C09107=1075.584,103.581,430.931,173.685,24.123,154.241
C09108=1075.591,103.830,430.912,173.686,24.125,154.241
C09109=1075.596,104.079,430.894,173.688,24.128,154.241
C09110=1075.601,104.329,430.875,173.690,24.130,154.241
C09111=1075.608,104.578,430.856,173.691,24.133,154.242
C09112=1075.613,104.827,430.838,173.693,24.135,154.242
C09113=1075.618,105.077,430.818,173.695,24.138,154.242
C09114=1075.625,105.326,430.800,173.696,24.141,154.243
C09115=1075.630,105.576,430.781,173.697,24.143,154.243
C09116=1075.635,105.824,430.762,173.700,24.146,154.243
C09117=1075.642,106.074,430.744,173.701,24.148,154.244
C09118=1075.647,106.323,430.724,173.702,24.151,154.244
C09119=1075.653,106.572,430.705,173.705,24.153,154.244
C09120=1075.659,106.821,430.688,173.706,24.156,154.244
C09121=1075.664,107.071,430.668,173.707,24.158,154.245
C09122=1075.669,107.320,430.649,173.710,24.161,154.245
C09123=1075.676,107.569,430.631,173.711,24.163,154.245
C09124=1075.682,107.818,430.612,173.712,24.165,154.246
C09125=1075.687,108.068,430.592,173.715,24.168,154.246
C09126=1075.693,108.316,430.574,173.716,24.171,154.246
C09127=1075.699,108.565,430.555,173.717,24.173,154.246
C09128=1075.704,108.816,430.536,173.720,24.176,154.247
C09129=1075.711,109.065,430.518,173.721,24.178,154.247
C09130=1075.716,109.313,430.499,173.722,24.180,154.247
C09131=1075.721,109.563,430.479,173.724,24.183,154.247
C09132=1075.728,109.812,430.461,173.726,24.185,154.248
C09133=1075.733,110.061,430.442,173.727,24.188,154.248
C09134=1075.739,110.311,430.422,173.729,24.190,154.248
C09135=1075.745,110.559,430.404,173.731,24.193,154.249
C09136=1075.751,110.840,430.382,173.733,24.196,154.249
C09137=1075.758,111.122,430.360,173.735,24.199,154.249
C09138=1075.764,111.404,430.339,173.736,24.202,154.250
C09139=1075.771,111.686,430.318,173.739,24.204,154.250
C09140=1075.777,111.935,430.298,173.740,24.207,154.250
C09141=1075.782,112.184,430.280,173.742,24.210,154.250
C09142=1075.788,112.433,430.261,173.744,24.212,154.251
C09143=1075.794,112.682,430.242,173.745,24.214,154.251
C09144=1075.799,112.932,430.222,173.747,24.217,154.251
C09145=1075.805,113.181,430.203,173.749,24.219,154.252
C09146=1075.810,113.430,430.184,173.750,24.222,154.252
C09147=1075.817,113.679,430.166,173.752,24.224,154.252
C09148=1075.823,113.928,430.146,173.754,24.227,154.252
C09149=1075.828,114.177,430.126,173.755,24.229,154.253
C09150=1075.834,114.427,430.107,173.757,24.232,154.253
C09151=1075.839,114.676,430.088,173.758,24.235,154.253
C09152=1075.845,114.925,430.069,173.761,24.237,154.254
C09153=1075.850,115.174,430.050,173.762,24.240,154.254
C09154=1075.856,115.424,430.030,173.763,24.242,154.254
C09155=1075.861,115.673,430.012,173.766,24.245,154.254
C09156=1075.867,115.921,429.992,173.767,24.247,154.255
C09157=1075.873,116.171,429.972,173.768,24.250,154.255
C09158=1075.879,116.420,429.953,173.771,24.252,154.255
C09159=1075.884,116.670,429.934,173.772,24.255,154.256
C09160=1075.889,116.918,429.915,173.774,24.257,154.256
C09161=1075.895,117.167,429.895,173.776,24.260,154.256
C09162=1075.901,117.417,429.876,173.777,24.263,154.257
C09163=1075.906,117.666,429.856,173.779,24.265,154.257
C09164=1075.912,117.916,429.837,173.780,24.268,154.257
C09165=1075.917,118.164,429.817,173.783,24.270,154.257
C09166=1075.923,118.413,429.798,173.784,24.273,154.258
C09167=1075.928,118.663,429.779,173.785,24.275,154.258
C09168=1075.934,118.912,429.759,173.788,24.278,154.258
C09169=1075.940,119.161,429.739,173.789,24.280,154.259
C09170=1075.946,119.410,429.720,173.790,24.282,154.259
C09171=1075.952,119.660,429.701,173.793,24.285,154.259
C09172=1075.957,119.908,429.681,173.794,24.288,154.259
C09173=1075.963,120.157,429.662,173.796,24.290,154.260
C09174=1075.968,120.407,429.643,173.798,24.293,154.260
C09175=1075.973,120.657,429.623,173.799,24.295,154.260
C09176=1075.979,120.905,429.603,173.801,24.298,154.260
C09177=1075.985,121.155,429.584,173.803,24.300,154.261
C09178=1075.991,121.404,429.564,173.805,24.303,154.261
C09179=1075.997,121.653,429.545,173.806,24.305,154.261
C09180=1076.002,121.903,429.525,173.808,24.307,154.262
C09181=1076.008,122.151,429.506,173.810,24.310,154.262
C09182=1076.013,122.400,429.487,173.811,24.312,154.262
C09183=1076.019,122.649,429.467,173.814,24.315,154.262
C09184=1076.024,122.899,429.447,173.815,24.318,154.263
C09185=1076.030,123.148,429.428,173.817,24.320,154.263
C09186=1076.036,123.397,429.408,173.819,24.323,154.263
C09187=1076.042,123.646,429.388,173.820,24.325,154.264
C09188=1076.048,123.895,429.368,173.822,24.328,154.264
C09189=1076.053,124.145,429.349,173.824,24.330,154.264
C09190=1076.059,124.393,429.329,173.826,24.333,154.264
C09191=1076.064,124.643,429.309,173.827,24.335,154.265
C09192=1076.070,124.892,429.289,173.829,24.337,154.265
C09193=1076.076,125.141,429.270,173.831,24.340,154.265
C09194=1076.082,125.390,429.250,173.832,24.342,154.265
C09195=1076.088,125.640,429.231,173.835,24.345,154.266
C09196=1076.094,125.888,429.211,173.836,24.347,154.266
C09197=1076.099,126.138,429.191,173.838,24.350,154.266
C09198=1076.105,126.387,429.171,173.840,24.353,154.267
C09199=1076.110,126.636,429.152,173.841,24.355,154.267
C09200=1076.117,126.917,429.130,173.843,24.358,154.267
C09201=1076.123,127.199,429.107,173.846,24.360,154.267
C09202=1076.130,127.481,429.085,173.848,24.363,154.268
C09203=1076.136,127.761,429.063,173.849,24.366,154.268
C09204=1076.141,128.011,429.043,173.851,24.369,154.268
C09205=1076.147,128.260,429.023,173.853,24.371,154.269
C09206=1076.154,128.509,429.003,173.855,24.373,154.269
C09207=1076.160,128.759,428.983,173.856,24.375,154.269
C09208=1076.166,129.008,428.963,173.859,24.378,154.269
C09209=1076.171,129.257,428.943,173.860,24.381,154.270
C09210=1076.177,129.506,428.924,173.861,24.383,154.270
C09211=1076.183,129.755,428.904,173.864,24.386,154.270
C09212=1076.189,130.004,428.884,173.865,24.388,154.270
C09213=1076.194,130.253,428.864,173.867,24.391,154.271
C09214=1076.199,130.502,428.844,173.869,24.392,154.271
C09215=1076.205,130.751,428.824,173.871,24.395,154.271
C09216=1076.211,131.001,428.805,173.873,24.397,154.271
C09217=1076.217,131.249,428.785,173.875,24.400,154.272
C09218=1076.223,131.499,428.764,173.876,24.402,154.272
C09219=1076.229,131.748,428.744,173.879,24.405,154.272
C09220=1076.235,131.998,428.725,173.880,24.407,154.272
C09221=1076.241,132.246,428.705,173.881,24.409,154.273
C09222=1076.246,132.495,428.684,173.884,24.412,154.273
C09223=1076.252,132.744,428.664,173.885,24.414,154.273
C09224=1076.257,132.994,428.644,173.887,24.417,154.273
C09225=1076.263,133.243,428.624,173.889,24.419,154.274
C09226=1076.268,133.492,428.604,173.891,24.422,154.274
C09227=1076.274,133.741,428.584,173.892,24.424,154.274
C09228=1076.279,133.990,428.563,173.895,24.427,154.275
C09229=1076.285,134.239,428.544,173.896,24.430,154.275
C09230=1076.290,134.488,428.523,173.898,24.432,154.275
C09231=1076.297,134.738,428.503,173.900,24.435,154.275
C09232=1076.302,134.987,428.483,173.902,24.437,154.276
C09233=1076.308,135.236,428.463,173.903,24.440,154.276
C09234=1076.313,135.485,428.442,173.905,24.442,154.276
C09235=1076.319,135.734,428.422,173.907,24.444,154.276
C09236=1076.325,135.983,428.402,173.909,24.446,154.277
C09237=1076.330,136.232,428.382,173.911,24.449,154.277
C09238=1076.336,136.482,428.362,173.912,24.451,154.277
C09239=1076.342,136.731,428.341,173.915,24.454,154.277
C09240=1076.347,136.980,428.321,173.916,24.456,154.278
C09241=1076.353,137.229,428.301,173.918,24.459,154.278
C09242=1076.359,137.478,428.280,173.920,24.462,154.278
C09243=1076.365,137.727,428.260,173.922,24.464,154.279
C09244=1076.370,137.976,428.240,173.923,24.466,154.279
C09245=1076.376,138.225,428.220,173.926,24.469,154.279
C09246=1076.382,138.475,428.199,173.927,24.471,154.279
C09247=1076.388,138.724,428.179,173.929,24.474,154.280
C09248=1076.393,138.973,428.158,173.931,24.476,154.280
C09249=1076.399,139.221,428.138,173.933,24.479,154.280
C09250=1076.404,139.471,428.118,173.934,24.481,154.280
C09251=1076.410,139.720,428.097,173.937,24.484,154.281
C09252=1076.416,139.969,428.077,173.938,24.486,154.281
C09253=1076.421,140.218,428.057,173.940,24.488,154.281
C09254=1076.427,140.467,428.037,173.942,24.491,154.281
C09255=1076.433,140.716,428.016,173.944,24.493,154.282
C09256=1076.438,140.965,427.995,173.945,24.496,154.282
C09257=1076.444,141.215,427.974,173.948,24.498,154.282
C09258=1076.450,141.463,427.954,173.949,24.501,154.282
C09259=1076.455,141.713,427.933,173.951,24.503,154.283
C09260=1076.461,141.962,427.913,173.953,24.506,154.283
C09261=1076.467,142.210,427.893,173.955,24.508,154.283
C09262=1076.472,142.460,427.872,173.956,24.511,154.284
C09263=1076.478,142.709,427.851,173.959,24.513,154.284
C09264=1076.484,142.990,427.828,173.961,24.516,154.284
C09265=1076.491,143.271,427.804,173.963,24.519,154.284
C09266=1076.497,143.552,427.781,173.965,24.521,154.285
C09267=1076.503,143.834,427.758,173.967,24.524,154.285
C09268=1076.509,144.083,427.738,173.969,24.527,154.285
C09269=1076.515,144.333,427.717,173.971,24.529,154.285
C09270=1076.520,144.582,427.696,173.973,24.532,154.286
C09271=1076.526,144.830,427.675,173.974,24.534,154.286
C09272=1076.532,145.079,427.655,173.977,24.537,154.286
C09273=1076.538,145.329,427.634,173.978,24.539,154.287
C09274=1076.543,145.578,427.614,173.980,24.542,154.287
C09275=1076.548,145.827,427.592,173.982,24.543,154.287
C09276=1076.554,146.076,427.572,173.984,24.546,154.287
C09277=1076.560,146.325,427.551,173.986,24.549,154.288
C09278=1076.566,146.574,427.530,173.988,24.551,154.288
C09279=1076.571,146.823,427.510,173.990,24.554,154.288
C09280=1076.577,147.073,427.489,173.992,24.556,154.288
C09281=1076.583,147.321,427.468,173.994,24.558,154.288
C09282=1076.588,147.570,427.448,173.995,24.561,154.289
C09283=1076.594,147.820,427.427,173.998,24.563,154.289
C09284=1076.600,148.068,427.405,173.999,24.566,154.289
C09285=1076.605,148.318,427.385,174.001,24.568,154.290
C09286=1076.610,148.567,427.364,174.003,24.571,154.290
C09287=1076.617,148.816,427.343,174.005,24.573,154.290
C09288=1076.623,149.065,427.323,174.007,24.575,154.290
C09289=1076.628,149.313,427.301,174.009,24.578,154.291
C09290=1076.634,149.563,427.280,174.011,24.581,154.291
C09291=1076.639,149.812,427.260,174.013,24.583,154.291
C09292=1076.645,150.061,427.239,174.015,24.586,154.291
C09293=1076.651,150.310,427.218,174.016,24.588,154.292
C09294=1076.656,150.559,427.196,174.019,24.590,154.292
C09295=1076.661,150.808,427.176,174.020,24.592,154.292
C09296=1076.668,151.057,427.154,174.022,24.595,154.292
C09297=1076.673,151.306,427.134,174.025,24.598,154.293
C09298=1076.678,151.555,427.112,174.026,24.600,154.293
C09299=1076.684,151.805,427.091,174.028,24.603,154.293
C09300=1076.690,152.053,427.070,174.030,24.605,154.293
C09301=1076.695,152.302,427.050,174.032,24.607,154.294
C09302=1076.701,152.552,427.028,174.034,24.610,154.294
C09303=1076.707,152.801,427.007,174.036,24.612,154.294
C09304=1076.712,153.049,426.986,174.038,24.615,154.294
C09305=1076.718,153.299,426.965,174.040,24.617,154.295
C09306=1076.724,153.548,426.944,174.042,24.620,154.295
C09307=1076.730,153.797,426.922,174.043,24.622,154.295
C09308=1076.735,154.046,426.902,174.046,24.624,154.295
C09309=1076.741,154.294,426.881,174.047,24.627,154.296
C09310=1076.746,154.544,426.860,174.049,24.629,154.296
C09311=1076.752,154.793,426.838,174.052,24.632,154.296
C09312=1076.758,155.042,426.817,174.053,24.634,154.297
C09313=1076.763,155.291,426.796,174.055,24.637,154.297
C09314=1076.769,155.540,426.775,174.057,24.639,154.297
C09315=1076.774,155.789,426.753,174.059,24.642,154.297
C09316=1076.780,156.038,426.732,174.061,24.644,154.297
C09317=1076.786,156.287,426.710,174.063,24.647,154.298
C09318=1076.791,156.536,426.689,174.065,24.649,154.298
C09319=1076.797,156.785,426.669,174.067,24.651,154.298
C09320=1076.803,157.034,426.647,174.069,24.654,154.298
C09321=1076.808,157.283,426.626,174.071,24.656,154.299
C09322=1076.814,157.532,426.604,174.073,24.659,154.299
C09323=1076.819,157.781,426.583,174.075,24.661,154.299
C09324=1076.825,158.031,426.561,174.076,24.664,154.300
C09325=1076.831,158.279,426.540,174.079,24.666,154.300
C09326=1076.837,158.528,426.518,174.081,24.669,154.300
C09327=1076.842,158.777,426.498,174.083,24.671,154.300
C09328=1076.848,159.059,426.473,174.085,24.674,154.301
C09329=1076.855,159.339,426.449,174.087,24.676,154.301
C09330=1076.861,159.620,426.425,174.089,24.679,154.301
C09331=1076.868,159.902,426.401,174.092,24.682,154.301
C09332=1076.873,160.150,426.379,174.094,24.684,154.302
C09333=1076.879,160.399,426.358,174.095,24.687,154.302
C09334=1076.884,160.648,426.336,174.098,24.689,154.302
C09335=1076.890,160.898,426.315,174.100,24.692,154.302
C09336=1076.896,161.146,426.294,174.101,24.694,154.303
C09337=1076.902,161.396,426.272,174.104,24.696,154.303
C09338=1076.906,161.644,426.250,174.106,24.699,154.303
C09339=1076.913,161.894,426.229,174.108,24.701,154.303
C09340=1076.917,162.142,426.207,174.110,24.704,154.304
C09341=1076.924,162.392,426.185,174.111,24.706,154.304
C09342=1076.928,162.640,426.163,174.114,24.709,154.304
C09343=1076.935,162.890,426.142,174.116,24.712,154.304
C09344=1076.939,163.138,426.120,174.117,24.714,154.305
C09345=1076.946,163.388,426.098,174.120,24.717,154.305
C09346=1076.950,163.636,426.076,174.122,24.719,154.305
C09347=1076.956,163.885,426.055,174.123,24.722,154.306
C09348=1076.961,164.135,426.033,174.126,24.724,154.306
C09349=1076.967,164.383,426.011,174.128,24.727,154.306
C09350=1076.972,164.633,425.989,174.129,24.729,154.306
C09351=1076.978,164.881,425.968,174.132,24.732,154.307
C09352=1076.983,165.131,425.946,174.134,24.734,154.307
C09353=1076.989,165.379,425.924,174.136,24.736,154.307
C09354=1076.994,165.629,425.902,174.138,24.739,154.307
C09355=1077.000,165.877,425.881,174.140,24.742,154.308
C09356=1077.005,166.127,425.859,174.142,24.744,154.308
C09357=1077.011,166.375,425.837,174.144,24.747,154.308
C09358=1077.016,166.625,425.815,174.146,24.749,154.308
C09359=1077.021,166.873,425.793,174.148,24.752,154.309
C09360=1077.028,167.122,425.771,174.150,24.754,154.309
C09361=1077.033,167.372,425.749,174.152,24.757,154.309
C09362=1077.039,167.620,425.727,174.154,24.759,154.309
C09363=1077.044,167.870,425.705,174.156,24.762,154.310
C09364=1077.050,168.118,425.684,174.158,24.764,154.310
C09365=1077.055,168.368,425.662,174.160,24.767,154.310
C09366=1077.060,168.616,425.640,174.162,24.769,154.310
C09367=1077.066,168.865,425.618,174.164,24.772,154.311
C09368=1077.072,169.114,425.595,174.166,24.774,154.311
C09369=1077.077,169.363,425.574,174.168,24.776,154.311
C09370=1077.083,169.613,425.552,174.171,24.779,154.311
C09371=1077.089,169.860,425.530,174.172,24.781,154.312
C09372=1077.094,170.110,425.508,174.174,24.784,154.312
C09373=1077.099,170.359,425.485,174.177,24.787,154.312
C09374=1077.105,170.608,425.464,174.179,24.789,154.313
C09375=1077.111,170.857,425.441,174.180,24.791,154.313
C09376=1077.116,171.105,425.420,174.183,24.794,154.313
C09377=1077.122,171.355,425.398,174.185,24.796,154.313
C09378=1077.127,171.604,425.375,174.186,24.799,154.314
C09379=1077.133,171.852,425.353,174.189,24.801,154.314
C09380=1077.138,172.102,425.331,174.191,24.804,154.314
C09381=1077.144,172.351,425.309,174.193,24.806,154.314
C09382=1077.150,172.599,425.287,174.195,24.809,154.314
C09383=1077.155,172.849,425.265,174.197,24.811,154.315
C09384=1077.162,173.097,425.242,174.200,24.814,154.315
C09385=1077.166,173.346,425.221,174.201,24.816,154.315
C09386=1077.172,173.596,425.198,174.203,24.818,154.315
C09387=1077.178,173.844,425.176,174.206,24.821,154.316
C09388=1077.184,174.094,425.154,174.207,24.823,154.316
C09389=1077.189,174.342,425.131,174.209,24.826,154.316
C09390=1077.195,174.591,425.110,174.212,24.829,154.317
C09391=1077.201,174.841,425.087,174.214,24.831,154.317
C09392=1077.206,175.121,425.062,174.216,24.834,154.317
C09393=1077.213,175.401,425.037,174.219,24.837,154.317
C09394=1077.219,175.682,425.011,174.221,24.839,154.318
C09395=1077.226,175.963,424.987,174.223,24.842,154.318
C09396=1077.232,176.212,424.964,174.226,24.845,154.318
C09397=1077.237,176.460,424.942,174.228,24.847,154.318
C09398=1077.242,176.710,424.920,174.230,24.849,154.319
C09399=1077.249,176.958,424.897,174.232,24.852,154.319
C09400=1077.254,177.208,424.875,174.234,24.854,154.319
C09401=1077.260,177.457,424.852,174.236,24.856,154.319
C09402=1077.266,177.705,424.831,174.238,24.859,154.319
C09403=1077.271,177.954,424.808,174.240,24.861,154.320
C09404=1077.277,178.204,424.786,174.243,24.864,154.320
C09405=1077.283,178.452,424.763,174.245,24.866,154.320
C09406=1077.289,178.701,424.740,174.247,24.869,154.320
C09407=1077.294,178.950,424.718,174.249,24.871,154.321
C09408=1077.299,179.199,424.695,174.251,24.874,154.321
C09409=1077.306,179.448,424.674,174.254,24.876,154.321
C09410=1077.311,179.697,424.651,174.255,24.878,154.321
C09411=1077.317,179.946,424.628,174.257,24.881,154.322
C09412=1077.323,180.195,424.606,174.260,24.884,154.322
C09413=1077.328,180.443,424.584,174.262,24.886,154.322
C09414=1077.334,180.692,424.561,174.264,24.888,154.322
C09415=1077.340,180.942,424.539,174.266,24.891,154.323
C09416=1077.345,181.191,424.516,174.268,24.893,154.323
C09417=1077.352,181.439,424.493,174.271,24.895,154.323
C09418=1077.357,181.688,424.470,174.273,24.898,154.323
C09419=1077.363,181.938,424.448,174.275,24.900,154.323
C09420=1077.369,182.187,424.425,174.277,24.903,154.324
C09421=1077.375,182.434,424.403,174.279,24.905,154.324
C09422=1077.380,182.683,424.380,174.282,24.908,154.324
C09423=1077.386,182.933,424.358,174.284,24.910,154.324
C09424=1077.391,183.182,424.335,174.285,24.912,154.325
C09425=1077.397,183.431,424.312,174.288,24.915,154.325
C09426=1077.404,183.679,424.290,174.290,24.917,154.325
C09427=1077.409,183.928,424.267,174.293,24.920,154.325
C09428=1077.415,184.178,424.245,174.295,24.922,154.326
C09429=1077.420,184.427,424.222,174.296,24.924,154.326
C09430=1077.426,184.675,424.199,174.299,24.927,154.326
C09431=1077.433,184.924,424.176,174.301,24.929,154.326
C09432=1077.438,185.173,424.153,174.303,24.932,154.327
C09433=1077.443,185.421,424.130,174.306,24.935,154.327
C09434=1077.449,185.670,424.107,174.307,24.937,154.327
C09435=1077.454,185.919,424.084,174.310,24.939,154.327
C09436=1077.460,186.169,424.062,174.312,24.942,154.328
C09437=1077.465,186.418,424.039,174.314,24.945,154.328
C09438=1077.470,186.667,424.016,174.317,24.947,154.328
C09439=1077.476,186.915,423.993,174.318,24.949,154.328
C09440=1077.481,187.164,423.970,174.320,24.952,154.329
C09441=1077.487,187.413,423.947,174.323,24.955,154.329
C09442=1077.493,187.662,423.924,174.325,24.957,154.329
C09443=1077.498,187.911,423.901,174.327,24.960,154.329
C09444=1077.503,188.160,423.878,174.330,24.963,154.330
C09445=1077.509,188.409,423.855,174.331,24.965,154.330
C09446=1077.515,188.658,423.832,174.334,24.967,154.330
C09447=1077.519,188.906,423.809,174.336,24.970,154.330
C09448=1077.525,189.155,423.786,174.338,24.972,154.331
C09449=1077.531,189.403,423.762,174.341,24.975,154.331
C09450=1077.537,189.652,423.739,174.343,24.978,154.331
C09451=1077.543,189.901,423.716,174.345,24.980,154.331
C09452=1077.548,190.150,423.693,174.347,24.983,154.332
C09453=1077.553,190.399,423.670,174.349,24.985,154.332
C09454=1077.559,190.648,423.647,174.351,24.988,154.332
C09455=1077.565,190.897,423.624,174.354,24.990,154.332
C09456=1077.571,191.177,423.597,174.356,24.993,154.333
C09457=1077.577,191.458,423.571,174.358,24.996,154.333
C09458=1077.583,191.739,423.545,174.362,24.999,154.333
C09459=1077.589,192.018,423.519,174.364,25.002,154.334
C09460=1077.594,192.267,423.496,174.366,25.004,154.334
C09461=1077.600,192.516,423.473,174.369,25.007,154.334
C09462=1077.606,192.764,423.449,174.370,25.009,154.334
C09463=1077.612,193.013,423.426,174.372,25.012,154.335
C09464=1077.617,193.262,423.402,174.375,25.014,154.335
C09465=1077.623,193.511,423.380,174.377,25.017,154.335
C09466=1077.629,193.760,423.355,174.379,25.019,154.335
C09467=1077.634,194.010,423.332,174.382,25.022,154.336
C09468=1077.640,194.258,423.309,174.384,25.025,154.336
C09469=1077.646,194.507,423.286,174.386,25.027,154.336
C09470=1077.651,194.756,423.262,174.389,25.030,154.336
C09471=1077.657,195.005,423.239,174.390,25.032,154.337
C09472=1077.662,195.254,423.216,174.392,25.035,154.337
C09473=1077.668,195.502,423.192,174.395,25.037,154.337
C09474=1077.673,195.751,423.169,174.397,25.039,154.337
C09475=1077.679,196.000,423.146,174.400,25.042,154.338
C09476=1077.685,196.248,423.122,174.402,25.045,154.338
C09477=1077.690,196.498,423.099,174.404,25.047,154.338
C09478=1077.696,196.747,423.076,174.407,25.050,154.338
C09479=1077.701,196.995,423.051,174.409,25.052,154.339
C09480=1077.707,197.244,423.028,174.411,25.055,154.339
C09481=1077.714,197.493,423.004,174.413,25.057,154.339
C09482=1077.719,197.742,422.981,174.415,25.060,154.339
C09483=1077.725,197.990,422.957,174.418,25.062,154.340
C09484=1077.730,198.239,422.934,174.420,25.064,154.340
C09485=1077.735,198.489,422.911,174.422,25.067,154.340
C09486=1077.741,198.737,422.887,174.425,25.070,154.340
C09487=1077.747,198.986,422.864,174.427,25.072,154.341
C09488=1077.753,199.235,422.839,174.429,25.075,154.341
C09489=1077.759,199.484,422.817,174.432,25.078,154.341
C09490=1077.764,199.733,422.792,174.434,25.080,154.341
C09491=1077.770,199.981,422.769,174.437,25.082,154.342
C09492=1077.776,200.230,422.746,174.439,25.085,154.342
C09493=1077.781,200.478,422.721,174.441,25.088,154.342
C09494=1077.787,200.728,422.698,174.444,25.090,154.342
C09495=1077.793,200.976,422.674,174.446,25.092,154.343
C09496=1077.798,201.225,422.651,174.447,25.095,154.343
C09497=1077.805,201.474,422.627,174.450,25.097,154.343
C09498=1077.810,201.723,422.604,174.452,25.100,154.343
C09499=1077.816,201.972,422.580,174.454,25.103,154.344
C09500=1077.821,202.220,422.555,174.457,25.105,154.344
C09501=1077.827,202.469,422.532,174.459,25.107,154.344
C09502=1077.832,202.718,422.508,174.462,25.110,154.344
C09503=1077.839,202.967,422.484,174.464,25.113,154.345
C09504=1077.844,203.216,422.461,174.466,25.115,154.345
C09505=1077.849,203.465,422.436,174.469,25.118,154.345
C09506=1077.855,203.713,422.413,174.471,25.121,154.345
C09507=1077.860,203.962,422.389,174.473,25.123,154.346
C09508=1077.866,204.211,422.365,174.476,25.126,154.346
C09509=1077.872,204.460,422.341,174.478,25.129,154.346
C09510=1077.878,204.708,422.317,174.480,25.131,154.346
C09511=1077.883,204.958,422.293,174.483,25.134,154.347
C09512=1077.889,205.206,422.269,174.485,25.136,154.347
C09513=1077.895,205.455,422.245,174.487,25.139,154.347
C09514=1077.900,205.704,422.221,174.490,25.141,154.347
C09515=1077.906,205.952,422.197,174.492,25.144,154.348
C09516=1077.911,206.201,422.173,174.495,25.146,154.348
C09517=1077.916,206.450,422.149,174.497,25.149,154.348
C09518=1077.922,206.699,422.124,174.499,25.152,154.348
C09519=1077.928,206.947,422.101,174.502,25.154,154.349
C09520=1077.956,208.196,421.979,174.611,25.215,154.348
C09521=1077.962,208.408,421.958,174.614,25.218,154.349
C09522=1077.967,208.620,421.937,174.616,25.221,154.349
C09523=1077.971,208.832,421.917,174.617,25.224,154.349
C09524=1077.976,209.045,421.895,174.619,25.227,154.350
C09525=1077.981,209.257,421.874,174.621,25.230,154.350
C09526=1077.986,209.470,421.853,174.623,25.233,154.351
C09527=1077.991,209.681,421.832,174.625,25.236,154.351
C09528=1077.997,209.931,421.807,174.627,25.239,154.352
C09529=1078.002,210.180,421.783,174.629,25.243,154.352
C09530=1078.008,210.428,421.758,174.631,25.247,154.353
C09531=1078.014,210.677,421.733,174.633,25.250,154.353
C09532=1078.020,210.925,421.708,174.636,25.254,154.354
C09533=1078.025,211.175,421.683,174.639,25.258,154.354
C09534=1078.030,211.423,421.658,174.641,25.261,154.354
C09535=1078.036,211.672,421.633,174.643,25.264,154.355
C09536=1078.042,211.920,421.608,174.645,25.268,154.356
C09537=1078.048,212.169,421.584,174.647,25.271,154.356
C09538=1078.053,212.417,421.559,174.649,25.275,154.356
C09539=1078.059,212.667,421.534,174.651,25.279,154.357
C09540=1078.065,212.915,421.509,174.654,25.282,154.357
C09541=1078.071,213.164,421.485,174.656,25.285,154.358
C09542=1078.076,213.413,421.459,174.659,25.289,154.358
C09543=1078.082,213.661,421.434,174.661,25.293,154.359
C09544=1078.088,213.910,421.409,174.663,25.296,154.359
C09545=1078.094,214.159,421.384,174.665,25.300,154.360
C09546=1078.098,214.408,421.359,174.667,25.304,154.360
C09547=1078.105,214.656,421.333,174.669,25.307,154.361
C09548=1078.110,214.904,421.309,174.671,25.310,154.361
C09549=1078.116,215.154,421.284,174.673,25.314,154.362
C09550=1078.122,215.402,421.258,174.676,25.318,154.362
C09551=1078.127,215.650,421.233,174.679,25.321,154.363
C09552=1078.133,215.900,421.208,174.681,25.325,154.363
C09553=1078.139,216.148,421.183,174.683,25.329,154.364
C09554=1078.144,216.397,421.157,174.685,25.332,154.364
C09555=1078.150,216.646,421.133,174.687,25.335,154.365
C09556=1078.156,216.894,421.108,174.689,25.339,154.365
C09557=1078.162,217.143,421.083,174.692,25.343,154.366
C09558=1078.167,217.392,421.057,174.695,25.346,154.366
C09559=1078.173,217.640,421.032,174.697,25.350,154.367
C09560=1078.178,217.878,421.007,174.699,25.353,154.367
C09561=1078.184,218.117,420.984,174.701,25.357,154.368
C09562=1078.189,218.356,420.960,174.703,25.360,154.368
C09563=1078.195,218.594,420.935,174.705,25.363,154.368
C09564=1078.201,218.834,420.910,174.707,25.367,154.369
C09565=1078.206,219.072,420.887,174.710,25.370,154.369
C09566=1078.212,219.311,420.862,174.712,25.373,154.370
C09567=1078.217,219.550,420.837,174.714,25.377,154.370
C09568=1078.223,219.797,420.812,174.716,25.380,154.371
C09569=1078.229,220.046,420.787,174.718,25.384,154.371
C09570=1078.234,220.295,420.761,174.721,25.387,154.372
C09571=1078.241,220.544,420.736,174.723,25.391,154.372
C09572=1078.246,220.792,420.712,174.726,25.395,154.373
C09573=1078.251,221.041,420.686,174.728,25.398,154.373
C09574=1078.258,221.290,420.660,174.730,25.401,154.374
C09575=1078.264,221.539,420.635,174.732,25.405,154.374
C09576=1078.273,221.947,420.593,174.737,25.411,154.375
C09577=1078.282,222.356,420.550,174.740,25.417,154.376
C09578=1078.291,222.764,420.508,174.744,25.423,154.376
C09579=1078.300,223.173,420.467,174.747,25.428,154.377
C09580=1078.306,223.422,420.441,174.749,25.432,154.378
C09581=1078.312,223.671,420.416,174.752,25.436,154.378
C09582=1078.318,223.920,420.390,174.755,25.439,154.379
C09583=1078.323,224.167,420.364,174.757,25.443,154.379
C09584=1078.329,224.416,420.338,174.759,25.446,154.380
C09585=1078.335,224.665,420.313,174.761,25.450,154.380
C09586=1078.341,224.914,420.287,174.764,25.453,154.381
C09587=1078.346,225.163,420.261,174.766,25.457,154.381
C09588=1078.352,225.411,420.236,174.768,25.461,154.382
C09589=1078.357,225.660,420.210,174.771,25.464,154.382
C09590=1078.364,225.908,420.184,174.773,25.467,154.383
C09591=1078.369,226.157,420.158,174.776,25.471,154.383
C09592=1078.375,226.406,420.132,174.778,25.474,154.383
C09593=1078.381,226.654,420.107,174.780,25.478,154.384
C09594=1078.386,226.903,420.081,174.782,25.482,154.384
C09595=1078.392,227.151,420.055,174.784,25.485,154.385
C09596=1078.398,227.400,420.029,174.787,25.489,154.385
C09597=1078.403,227.649,420.003,174.790,25.493,154.386
C09598=1078.410,227.897,419.977,174.792,25.496,154.386
C09599=1078.415,228.146,419.951,174.794,25.499,154.387
C09600=1078.421,228.395,419.925,174.796,25.502,154.387
C09601=1078.427,228.643,419.900,174.799,25.506,154.388
C09602=1078.433,228.892,419.873,174.801,25.510,154.388
C09603=1078.439,229.140,419.848,174.804,25.513,154.389
C09604=1078.444,229.389,419.822,174.806,25.517,154.389
C09605=1078.449,229.637,419.796,174.809,25.521,154.390
C09606=1078.456,229.886,419.770,174.811,25.524,154.390
C09607=1078.461,230.134,419.744,174.813,25.528,154.391
C09608=1078.467,230.383,419.718,174.815,25.531,154.391
C09609=1078.472,230.632,419.692,174.818,25.535,154.392
C09610=1078.478,230.880,419.665,174.820,25.538,154.392
C09611=1078.484,231.129,419.640,174.823,25.542,154.393
C09612=1078.490,231.377,419.613,174.825,25.545,154.393
C09613=1078.496,231.626,419.587,174.827,25.549,154.394
C09614=1078.501,231.875,419.561,174.830,25.553,154.394
C09615=1078.507,232.124,419.535,174.832,25.556,154.394
C09616=1078.513,232.372,419.508,174.834,25.559,154.395
C09617=1078.519,232.621,419.483,174.836,25.563,154.395
C09618=1078.525,232.869,419.456,174.840,25.567,154.396
C09619=1078.530,233.118,419.430,174.842,25.570,154.396
C09620=1078.536,233.366,419.403,174.844,25.574,154.397
C09621=1078.542,233.615,419.377,174.846,25.577,154.397
C09622=1078.547,233.864,419.351,174.849,25.581,154.398
C09623=1078.553,234.112,419.324,174.851,25.585,154.398
C09624=1078.558,234.360,419.299,174.853,25.588,154.399
C09625=1078.563,234.609,419.272,174.856,25.591,154.399
C09626=1078.569,234.857,419.245,174.859,25.595,154.400
C09627=1078.575,235.106,419.219,174.861,25.599,154.400
C09628=1078.584,235.507,419.177,174.864,25.604,154.401
C09629=1078.593,235.906,419.134,174.868,25.610,154.402
C09630=1078.603,236.306,419.092,174.873,25.616,154.403
C09631=1078.613,236.707,419.049,174.876,25.622,154.403
C09632=1078.618,236.956,419.022,174.878,25.625,154.404
C09633=1078.624,237.205,418.996,174.882,25.629,154.404
C09634=1078.630,237.453,418.970,174.884,25.632,154.405
C09635=1078.635,237.701,418.943,174.886,25.636,154.405
C09636=1078.641,237.950,418.916,174.888,25.639,154.406
C09637=1078.646,238.198,418.889,174.891,25.643,154.406
C09638=1078.652,238.447,418.863,174.893,25.647,154.407
C09639=1078.657,238.696,418.836,174.895,25.650,154.407
C09640=1078.663,238.944,418.810,174.898,25.654,154.408
C09641=1078.669,239.193,418.783,174.901,25.657,154.408
C09642=1078.675,239.441,418.757,174.903,25.661,154.409
C09643=1078.681,239.690,418.730,174.905,25.664,154.409
C09644=1078.687,239.938,418.703,174.908,25.668,154.410
C09645=1078.693,240.187,418.676,174.910,25.671,154.410
C09646=1078.699,240.435,418.650,174.912,25.675,154.411
C09647=1078.704,240.684,418.624,174.916,25.679,154.411
C09648=1078.710,240.932,418.597,174.918,25.682,154.411
C09649=1078.716,241.181,418.570,174.920,25.686,154.412
C09650=1078.721,241.429,418.543,174.922,25.689,154.412
C09651=1078.727,241.678,418.516,174.925,25.693,154.413
C09652=1078.733,241.927,418.489,174.927,25.696,154.413
C09653=1078.738,242.175,418.463,174.930,25.699,154.414
C09654=1078.744,242.424,418.436,174.933,25.703,154.414
C09655=1078.750,242.671,418.409,174.935,25.707,154.415
C09656=1078.757,242.920,418.382,174.937,25.710,154.415
C09657=1078.762,243.169,418.355,174.940,25.714,154.416
C09658=1078.768,243.417,418.328,174.942,25.718,154.416
C09659=1078.773,243.666,418.301,174.944,25.721,154.417
C09660=1078.778,243.914,418.274,174.948,25.725,154.417
C09661=1078.784,244.163,418.247,174.950,25.728,154.418
C09662=1078.790,244.412,418.220,174.952,25.732,154.418
C09663=1078.796,244.661,418.193,174.955,25.736,154.419
C09664=1078.802,244.908,418.166,174.957,25.739,154.419
C09665=1078.807,245.157,418.139,174.959,25.743,154.420
C09666=1078.812,245.405,418.112,174.961,25.746,154.420
C09667=1078.818,245.654,418.085,174.965,25.750,154.421
C09668=1078.825,245.903,418.058,174.967,25.753,154.421
C09669=1078.830,246.151,418.030,174.969,25.757,154.422
C09670=1078.836,246.399,418.004,174.972,25.761,154.422
C09671=1078.841,246.647,417.977,174.974,25.764,154.423
C09672=1078.847,246.896,417.949,174.976,25.768,154.423
C09673=1078.853,247.145,417.922,174.979,25.772,154.424
C09674=1078.858,247.393,417.895,174.982,25.775,154.424
C09675=1078.864,247.642,417.868,174.985,25.779,154.424
C09676=1078.870,247.890,417.840,174.987,25.782,154.425
C09677=1078.876,248.139,417.813,174.989,25.786,154.426
C09678=1078.881,248.387,417.785,174.992,25.790,154.426
C09679=1078.886,248.635,417.758,174.994,25.793,154.427
C09680=1078.896,249.029,417.714,174.998,25.799,154.427
C09681=1078.905,249.423,417.672,175.003,25.805,154.428
C09682=1078.913,249.816,417.628,175.006,25.811,154.429
C09683=1078.923,250.210,417.585,175.010,25.816,154.430
C09684=1078.928,250.458,417.557,175.013,25.820,154.430
C09685=1078.933,250.707,417.530,175.015,25.824,154.431
C09686=1078.940,250.955,417.502,175.017,25.827,154.431
C09687=1078.945,251.204,417.475,175.021,25.831,154.432
C09688=1078.951,251.452,417.447,175.023,25.834,154.432
C09689=1078.956,251.700,417.420,175.025,25.838,154.433
C09690=1078.962,251.949,417.392,175.028,25.842,154.433
C09691=1078.968,252.197,417.365,175.030,25.845,154.434
C09692=1078.973,252.445,417.337,175.032,25.848,154.434
C09693=1078.979,252.694,417.309,175.035,25.852,154.435
C09694=1078.985,252.942,417.282,175.038,25.856,154.435
C09695=1078.991,253.191,417.254,175.041,25.860,154.436
C09696=1078.997,253.439,417.227,175.043,25.863,154.436
C09697=1079.002,253.688,417.199,175.045,25.867,154.437
C09698=1079.008,253.936,417.171,175.048,25.871,154.437
C09699=1079.014,254.184,417.144,175.050,25.874,154.438
C09700=1079.019,254.433,417.116,175.053,25.878,154.438
C09701=1079.025,254.682,417.088,175.056,25.881,154.439
C09702=1079.031,254.929,417.061,175.058,25.885,154.439
C09703=1079.036,255.179,417.033,175.061,25.889,154.440
C09704=1079.042,255.427,417.005,175.063,25.892,154.440
C09705=1079.048,255.674,416.978,175.066,25.896,154.440
C09706=1079.054,255.923,416.949,175.068,25.899,154.441
C09707=1079.059,256.172,416.922,175.071,25.903,154.442
C09708=1079.065,256.420,416.894,175.074,25.907,154.442
C09709=1079.071,256.668,416.866,175.076,25.910,154.442
C09710=1079.077,256.917,416.838,175.079,25.914,154.443
C09711=1079.082,257.165,416.810,175.081,25.917,154.444
C09712=1079.089,257.414,416.782,175.083,25.921,154.444
C09713=1079.094,257.662,416.755,175.087,25.924,154.444
C09714=1079.100,257.911,416.727,175.089,25.928,154.445
C09715=1079.106,258.159,416.700,175.092,25.932,154.445
C09716=1079.112,258.408,416.671,175.094,25.935,154.446
C09717=1079.117,258.656,416.643,175.096,25.939,154.446
C09718=1079.123,258.904,416.615,175.099,25.943,154.447
C09719=1079.129,259.152,416.588,175.101,25.946,154.447
C09720=1079.135,259.401,416.559,175.105,25.950,154.448
C09721=1079.140,259.649,416.531,175.107,25.953,154.448
C09722=1079.146,259.898,416.503,175.110,25.957,154.449
C09723=1079.152,260.145,416.476,175.112,25.960,154.449
C09724=1079.158,260.394,416.447,175.114,25.964,154.450
C09725=1079.164,260.643,416.419,175.117,25.968,154.450
C09726=1079.170,260.891,416.391,175.120,25.971,154.451
C09727=1079.176,261.139,416.363,175.123,25.975,154.451
C09728=1079.182,261.387,416.335,175.125,25.978,154.452
C09729=1079.188,261.636,416.307,175.128,25.982,154.452
C09730=1079.193,261.884,416.279,175.130,25.985,154.453
C09731=1079.199,262.133,416.251,175.134,25.989,154.453
C09732=1079.208,262.523,416.206,175.137,25.994,154.454
C09733=1079.218,262.914,416.162,175.141,26.000,154.455
C09734=1079.227,263.305,416.118,175.146,26.006,154.455
C09735=1079.237,263.696,416.073,175.149,26.012,154.456
C09736=1079.243,263.944,416.045,175.153,26.015,154.457
C09737=1079.249,264.193,416.017,175.155,26.019,154.457
C09738=1079.254,264.441,415.989,175.158,26.023,154.458
C09739=1079.260,264.689,415.960,175.160,26.026,154.458
C09740=1079.266,264.937,415.932,175.163,26.030,154.459
C09741=1079.272,265.186,415.903,175.165,26.033,154.459
C09742=1079.277,265.435,415.874,175.168,26.037,154.460
C09743=1079.282,265.683,415.846,175.171,26.041,154.460
C09744=1079.288,265.931,415.817,175.173,26.044,154.461
C09745=1079.294,266.179,415.789,175.176,26.048,154.461
C09746=1079.300,266.428,415.760,175.178,26.052,154.462
C09747=1079.306,266.676,415.732,175.181,26.056,154.462
C09748=1079.312,266.924,415.703,175.183,26.059,154.463
C09749=1079.317,267.173,415.675,175.187,26.063,154.463
C09750=1079.324,267.421,415.646,175.189,26.066,154.464
C09751=1079.328,267.669,415.617,175.192,26.070,154.464
C09752=1079.334,267.918,415.589,175.194,26.074,154.465
C09753=1079.341,268.166,415.560,175.197,26.078,154.465
C09754=1079.346,268.414,415.532,175.199,26.081,154.466
C09755=1079.352,268.662,415.503,175.202,26.085,154.466
C09756=1079.358,268.911,415.475,175.205,26.088,154.467
C09757=1079.364,269.159,415.446,175.208,26.092,154.467
C09758=1079.369,269.407,415.417,175.210,26.096,154.468
C09759=1079.375,269.655,415.388,175.213,26.100,154.468
C09760=1079.381,269.904,415.359,175.215,26.103,154.469
C09761=1079.387,270.152,415.331,175.218,26.107,154.469
C09762=1079.392,270.400,415.301,175.221,26.111,154.470
C09763=1079.398,270.649,415.273,175.224,26.115,154.470
C09764=1079.404,270.897,415.244,175.226,26.118,154.471
C09765=1079.410,271.144,415.215,175.229,26.121,154.471
C09766=1079.415,271.393,415.187,175.231,26.125,154.472
C09767=1079.422,271.642,415.157,175.234,26.129,154.472
C09768=1079.428,271.890,415.128,175.237,26.133,154.473
C09769=1079.432,272.138,415.100,175.240,26.136,154.473
C09770=1079.439,272.386,415.071,175.242,26.140,154.474
C09771=1079.445,272.634,415.042,175.245,26.144,154.474
C09772=1079.451,272.883,415.013,175.247,26.147,154.475
C09773=1079.456,273.131,414.984,175.250,26.151,154.475
C09774=1079.462,273.379,414.955,175.253,26.155,154.476
C09775=1079.468,273.627,414.926,175.256,26.159,154.477
C09776=1079.473,273.876,414.897,175.258,26.162,154.477
C09777=1079.480,274.124,414.868,175.261,26.166,154.478
C09778=1079.485,274.372,414.839,175.264,26.170,154.478
C09779=1079.491,274.620,414.810,175.266,26.173,154.478
C09780=1079.496,274.869,414.780,175.269,26.177,154.479
C09781=1079.503,275.117,414.751,175.272,26.181,154.480
C09782=1079.508,275.366,414.722,175.275,26.185,154.480
C09783=1079.513,275.613,414.694,175.277,26.188,154.481
C09784=1079.523,276.007,414.647,175.282,26.194,154.481
C09785=1079.532,276.401,414.601,175.285,26.200,154.482
C09786=1079.542,276.795,414.554,175.290,26.206,154.483
C09787=1079.550,277.189,414.507,175.295,26.212,154.484
C09788=1079.557,277.437,414.478,175.297,26.216,154.484
C09789=1079.562,277.685,414.449,175.300,26.220,154.485
C09790=1079.568,277.934,414.420,175.302,26.223,154.485
C09791=1079.573,278.181,414.390,175.305,26.227,154.486
C09792=1079.580,278.429,414.361,175.308,26.231,154.487
C09793=1079.585,278.678,414.332,175.311,26.235,154.487
C09794=1079.591,278.926,414.302,175.314,26.238,154.488
C09795=1079.597,279.175,414.273,175.316,26.242,154.488
C09796=1079.602,279.423,414.243,175.319,26.246,154.489
C09797=1079.609,279.671,414.214,175.321,26.249,154.489
C09798=1079.614,279.920,414.185,175.324,26.253,154.490
C09799=1079.621,280.167,414.155,175.327,26.257,154.490
C09800=1079.626,280.415,414.125,175.330,26.261,154.491
C09801=1079.632,280.664,414.096,175.333,26.265,154.491
C09802=1079.638,280.912,414.067,175.335,26.268,154.492
C09803=1079.644,281.161,414.037,175.338,26.272,154.492
C09804=1079.649,281.408,414.007,175.340,26.276,154.493
C09805=1079.654,281.656,413.977,175.343,26.280,154.493
C09806=1079.661,281.904,413.948,175.346,26.284,154.494
C09807=1079.666,282.153,413.919,175.349,26.287,154.494
C09808=1079.672,282.400,413.888,175.352,26.291,154.495
C09809=1079.677,282.649,413.859,175.354,26.295,154.496
C09810=1079.684,282.897,413.830,175.357,26.299,154.496
C09811=1079.689,283.145,413.799,175.360,26.303,154.497
C09812=1079.695,283.393,413.770,175.362,26.307,154.497
C09813=1079.700,283.642,413.740,175.365,26.311,154.498
C09814=1079.707,283.889,413.710,175.368,26.314,154.498
C09815=1079.713,284.138,413.681,175.371,26.318,154.499
C09816=1079.718,284.386,413.651,175.374,26.322,154.499
C09817=1079.724,284.634,413.621,175.376,26.325,154.500
C09818=1079.729,284.882,413.591,175.379,26.329,154.500
C09819=1079.735,285.130,413.561,175.381,26.333,154.501
C09820=1079.741,285.378,413.532,175.385,26.337,154.502
C09821=1079.747,285.626,413.501,175.388,26.341,154.502
C09822=1079.753,285.875,413.472,175.390,26.345,154.503
C09823=1079.759,286.122,413.441,175.393,26.348,154.503
C09824=1079.764,286.371,413.412,175.395,26.352,154.504
C09825=1079.770,286.619,413.381,175.398,26.356,154.504
C09826=1079.776,286.867,413.352,175.401,26.360,154.505
C09827=1079.782,287.115,413.322,175.404,26.364,154.505
C09828=1079.788,287.363,413.291,175.407,26.368,154.506
C09829=1079.794,287.612,413.261,175.410,26.372,154.506
C09830=1079.800,287.859,413.231,175.412,26.375,154.507
C09831=1079.805,288.108,413.202,175.415,26.379,154.507
C09832=1079.811,288.356,413.171,175.418,26.383,154.508
C09833=1079.818,288.603,413.141,175.420,26.387,154.509
C09834=1079.823,288.852,413.112,175.424,26.391,154.509
C09835=1079.829,289.099,413.081,175.426,26.394,154.510
C09836=1079.838,289.503,413.032,175.431,26.400,154.510
C09837=1079.847,289.907,412.983,175.435,26.407,154.511
C09838=1079.857,290.311,412.934,175.440,26.413,154.512
C09839=1079.867,290.715,412.884,175.444,26.420,154.513
C09840=1079.873,290.963,412.854,175.447,26.423,154.514
C09841=1079.879,291.211,412.824,175.450,26.428,154.514
C09842=1079.885,291.458,412.793,175.453,26.431,154.515
C09843=1079.889,291.707,412.763,175.456,26.435,154.515
C09844=1079.895,291.955,412.733,175.459,26.439,154.516
C09845=1079.902,292.204,412.702,175.461,26.443,154.517
C09846=1079.907,292.451,412.672,175.464,26.447,154.517
C09847=1079.913,292.699,412.641,175.467,26.451,154.518
C09848=1079.919,292.947,412.611,175.470,26.455,154.518
C09849=1079.925,293.195,412.581,175.473,26.459,154.519
C09850=1079.931,293.443,412.550,175.476,26.463,154.519
C09851=1079.937,293.691,412.520,175.478,26.467,154.520
C09852=1079.942,293.939,412.489,175.481,26.470,154.521
C09853=1079.948,294.187,412.458,175.484,26.474,154.521
C09854=1079.954,294.435,412.428,175.486,26.478,154.522
C09855=1079.960,294.683,412.397,175.490,26.482,154.522
C09856=1079.966,294.931,412.367,175.493,26.486,154.523
C09857=1079.972,295.179,412.337,175.495,26.490,154.523
C09858=1079.977,295.427,412.306,175.498,26.494,154.524
C09859=1079.983,295.676,412.275,175.501,26.498,154.524
C09860=1079.989,295.924,412.245,175.504,26.502,154.525
C09861=1079.995,296.171,412.214,175.506,26.506,154.526
C09862=1080.000,296.420,412.183,175.509,26.510,154.526
C09863=1080.007,296.667,412.152,175.513,26.514,154.527
C09864=1080.013,296.915,412.121,175.515,26.517,154.527
C09865=1080.018,297.163,412.091,175.518,26.522,154.528
C09866=1080.024,297.412,412.060,175.521,26.526,154.528
C09867=1080.030,297.660,412.029,175.523,26.530,154.529
C09868=1080.036,297.907,411.998,175.526,26.533,154.530
C09869=1080.041,298.155,411.967,175.529,26.538,154.530
C09870=1080.048,298.404,411.937,175.533,26.542,154.531
C09871=1080.053,298.652,411.906,175.535,26.546,154.531
C09872=1080.059,298.899,411.875,175.538,26.549,154.532
C09873=1080.064,299.147,411.844,175.541,26.554,154.533
C09874=1080.070,299.396,411.813,175.544,26.558,154.533
C09875=1080.076,299.643,411.781,175.546,26.562,154.534
C09876=1080.082,299.891,411.751,175.549,26.566,154.534
C09877=1080.087,300.139,411.720,175.552,26.570,154.535
C09878=1080.093,300.387,411.688,175.555,26.574,154.536
C09879=1080.098,300.635,411.658,175.558,26.578,154.536
C09880=1080.104,300.883,411.626,175.561,26.582,154.537
C09881=1080.110,301.131,411.595,175.564,26.586,154.537
C09882=1080.115,301.379,411.564,175.566,26.590,154.538
C09883=1080.121,301.626,411.533,175.569,26.594,154.539
C09884=1080.127,301.875,411.502,175.572,26.599,154.539
C09885=1080.133,302.122,411.471,175.575,26.603,154.540
C09886=1080.138,302.371,411.440,175.578,26.607,154.540
C09887=1080.144,302.619,411.408,175.581,26.611,154.541
C09888=1080.154,303.037,411.356,175.586,26.618,154.542
C09889=1080.164,303.454,411.303,175.591,26.625,154.543
C09890=1080.174,303.873,411.250,175.595,26.631,154.544
C09891=1080.184,304.291,411.197,175.601,26.639,154.545
C09892=1080.189,304.539,411.166,175.603,26.642,154.546
C09893=1080.195,304.787,411.134,175.606,26.646,154.546
C09894=1080.201,305.034,411.103,175.609,26.651,154.547
C09895=1080.206,305.282,411.072,175.612,26.655,154.548
C09896=1080.213,305.530,411.041,175.615,26.659,154.548
C09897=1080.218,305.778,411.009,175.617,26.663,154.549
C09898=1080.224,306.027,410.978,175.620,26.667,154.550
C09899=1080.230,306.274,410.947,175.624,26.671,154.550
C09900=1080.236,306.522,410.915,175.627,26.675,154.551
C09901=1080.241,306.770,410.883,175.630,26.680,154.551
C09902=1080.248,307.017,410.851,175.632,26.683,154.552
C09903=1080.253,307.266,410.821,175.635,26.688,154.553
C09904=1080.259,307.514,410.789,175.638,26.692,154.553
C09905=1080.265,307.761,410.757,175.641,26.696,154.554
C09906=1080.271,308.009,410.725,175.644,26.700,154.554
C09907=1080.277,308.257,410.693,175.647,26.704,154.555
C09908=1080.283,308.505,410.662,175.650,26.708,154.556
C09909=1080.289,308.753,410.630,175.653,26.712,154.556
C09910=1080.295,309.001,410.599,175.656,26.717,154.557
C09911=1080.301,309.249,410.567,175.659,26.721,154.557
C09912=1080.307,309.496,410.536,175.662,26.725,154.558
C09913=1080.313,309.745,410.504,175.664,26.729,154.559
C09914=1080.319,309.993,410.472,175.667,26.733,154.559
C09915=1080.324,310.240,410.441,175.671,26.737,154.560
C09916=1080.331,310.488,410.409,175.674,26.741,154.560
C09917=1080.337,310.736,410.377,175.677,26.746,154.561
C09918=1080.342,310.984,410.345,175.679,26.750,154.562
C09919=1080.348,311.232,410.313,175.682,26.754,154.562
C09920=1080.355,311.480,410.282,175.685,26.758,154.563
C09921=1080.361,311.727,410.250,175.688,26.762,154.564
C09922=1080.366,311.975,410.218,175.691,26.766,154.564
C09923=1080.372,312.223,410.186,175.694,26.771,154.565
C09924=1080.378,312.471,410.154,175.698,26.775,154.566
C09925=1080.385,312.719,410.122,175.700,26.778,154.566
C09926=1080.391,312.967,410.090,175.703,26.783,154.567
C09927=1080.397,313.215,410.058,175.706,26.787,154.567
C09928=1080.402,313.462,410.026,175.709,26.791,154.568
C09929=1080.408,313.710,409.994,175.712,26.796,154.569
C09930=1080.415,313.958,409.963,175.715,26.799,154.569
C09931=1080.421,314.206,409.931,175.718,26.804,154.570
C09932=1080.426,314.454,409.899,175.721,26.808,154.570
C09933=1080.433,314.702,409.866,175.724,26.812,154.571
C09934=1080.439,314.950,409.834,175.727,26.816,154.572
C09935=1080.445,315.198,409.802,175.730,26.821,154.572
C09936=1080.450,315.445,409.769,175.733,26.825,154.573
C09937=1080.456,315.693,409.737,175.736,26.829,154.574
C09938=1080.462,315.942,409.705,175.739,26.834,154.575
C09939=1080.467,316.188,409.673,175.741,26.838,154.575
C09940=1080.472,316.399,409.645,175.744,26.842,154.576
C09941=1080.477,316.610,409.617,175.747,26.845,154.576
C09942=1080.482,316.821,409.590,175.749,26.849,154.577
C09943=1080.487,317.031,409.563,175.752,26.853,154.577
C09944=1080.492,317.242,409.535,175.754,26.857,154.578
C09945=1080.496,317.453,409.507,175.757,26.860,154.579
C09946=1080.501,317.663,409.480,175.759,26.864,154.579
C09947=1080.506,317.873,409.453,175.762,26.868,154.580
C09948=1080.512,318.121,409.420,175.765,26.872,154.580
C09949=1080.518,318.369,409.388,175.768,26.877,154.581
C09950=1080.524,318.617,409.355,175.770,26.881,154.582
C09951=1080.529,318.864,409.323,175.773,26.885,154.582
C09952=1080.536,319.112,409.290,175.776,26.890,154.583
C09953=1080.541,319.361,409.258,175.780,26.894,154.584
C09954=1080.547,319.608,409.225,175.783,26.899,154.585
C09955=1080.553,319.856,409.192,175.786,26.903,154.585
C09956=1080.558,320.104,409.160,175.789,26.907,154.586
C09957=1080.564,320.351,409.127,175.792,26.912,154.587
C09958=1080.571,320.599,409.095,175.795,26.916,154.587
C09959=1080.576,320.847,409.062,175.798,26.921,154.588
C09960=1080.582,321.095,409.029,175.800,26.925,154.589
C09961=1080.588,321.343,408.996,175.803,26.930,154.589
C09962=1080.594,321.591,408.964,175.806,26.934,154.590
C09963=1080.599,321.838,408.931,175.809,26.938,154.591
C09964=1080.606,322.086,408.899,175.812,26.943,154.591
C09965=1080.611,322.333,408.865,175.816,26.947,154.592
C09966=1080.617,322.582,408.833,175.819,26.952,154.593
C09967=1080.623,322.830,408.800,175.822,26.956,154.594
C09968=1080.629,323.077,408.767,175.825,26.961,154.594
C09969=1080.635,323.325,408.734,175.828,26.965,154.595
C09970=1080.641,323.573,408.701,175.831,26.970,154.596
C09971=1080.647,323.821,408.669,175.834,26.974,154.596
C09972=1080.653,324.068,408.636,175.837,26.978,154.597
C09973=1080.659,324.316,408.603,175.840,26.983,154.598
C09974=1080.665,324.564,408.570,175.843,26.987,154.598
C09975=1080.671,324.812,408.537,175.846,26.992,154.599
C09976=1080.677,325.059,408.504,175.848,26.996,154.600
C09977=1080.682,325.307,408.471,175.852,27.000,154.600
C09978=1080.689,325.555,408.438,175.855,27.005,154.601
C09979=1080.695,325.803,408.405,175.858,27.009,154.602
C09980=1080.701,326.050,408.372,175.861,27.014,154.603
C09981=1080.707,326.298,408.339,175.864,27.019,154.603
C09982=1080.712,326.546,408.306,175.867,27.023,154.604
C09983=1080.719,326.794,408.273,175.870,27.028,154.605
C09984=1080.724,327.041,408.240,175.873,27.032,154.605
C09985=1080.731,327.289,408.207,175.876,27.037,154.606
C09986=1080.736,327.537,408.174,175.879,27.041,154.607
C09987=1080.742,327.785,408.141,175.882,27.046,154.608
C09988=1080.748,328.032,408.107,175.885,27.050,154.608
C09989=1080.755,328.279,408.074,175.888,27.055,154.609
C09990=1080.761,328.528,408.041,175.892,27.059,154.610
C09991=1080.767,328.776,408.008,175.895,27.064,154.610
C09992=1080.773,329.024,407.974,175.898,27.068,154.611
C09993=1080.779,329.271,407.942,175.901,27.073,154.612
C09994=1080.785,329.518,407.908,175.904,27.078,154.613
C09995=1080.791,329.766,407.875,175.907,27.082,154.613
C09996=1080.801,330.181,407.819,175.912,27.090,154.615
//INST
///DATE 2021/06/25 14:45
///ATTR SC,RW,RJ
////FRAME ROBOT
///GROUP1 RB1
NOP
MOVL C00000 V=800.0 PL=0
MOVL C00001 V=800.0 PL=0
MOVL C00002 V=800.0 PL=0
MOVL C00003 V=800.0 PL=0
MOVL C00004 V=800.0 PL=0
MOVL C00005 V=800.0 PL=0
MOVL C00006 V=800.0 PL=0
MOVL C00007 V=800.0 PL=0
MOVL C00008 V=800.0 PL=0
MOVL C00009 V=800.0 PL=0
MOVL C00010 V=800.0 PL=0
MOVL C00011 V=800.0 PL=0
MOVL C00012 V=800.0 PL=0
MOVL C00013 V=800.0 PL=0
MOVL C00014 V=800.0 PL=0
MOVL C00015 V=800.0 PL=0
MOVL C00016 V=800.0 PL=0
MOVL C00017 V=800.0 PL=0
MOVL C00018 V=800.0 PL=0
MOVL C00019 V=800.0 PL=0
MOVL C00020 V=800.0 PL=0
MOVL C00021 V=800.0 PL=0
MOVL C00022 V=800.0 PL=0
MOVL C00023 V=800.0 PL=0
MOVL C00024 V=800.0 PL=0
MOVL C00025 V=800.0 PL=0
MOVL C00026 V=800.0 PL=0
MOVL C00027 V=800.0 PL=0
MOVL C00028 V=800.0 PL=0
MOVL C00029 V=800.0 PL=0
MOVL C00030 V=800.0 PL=0
MOVL C00031 V=800.0 PL=0
MOVL C00032 V=800.0 PL=0
MOVL C00033 V=800.0 PL=0
MOVL C00034 V=800.0 PL=0
MOVL C00035 V=800.0 PL=0
MOVL C00036 V=800.0 PL=0
MOVL C00037 V=800.0 PL=0
MOVL C00038 V=800.0 PL=0
MOVL C00039 V=800.0 PL=0
MOVL C00040 V=800.0 PL=0
MOVL C00041 V=800.0 PL=0
MOVL C00042 V=800.0 PL=0
MOVL C00043 V=800.0 PL=0
MOVL C00044 V=800.0 PL=0
MOVL C00045 V=800.0 PL=0
MOVL C00046 V=800.0 PL=0
MOVL C00047 V=800.0 PL=0
MOVL C00048 V=800.0 PL=0
MOVL C00049 V=800.0 PL=0
MOVL C00050 V=800.0 PL=0
MOVL C00051 V=800.0 PL=0
MOVL C00052 V=800.0 PL=0
MOVL C00053 V=800.0 PL=0
MOVL C00054 V=800.0 PL=0
MOVL C00055 V=800.0 PL=0
MOVL C00056 V=800.0 PL=0
MOVL C00057 V=800.0 PL=0
MOVL C00058 V=800.0 PL=0
MOVL C00059 V=800.0 PL=0
MOVL C00060 V=800.0 PL=0
MOVL C00061 V=800.0 PL=0
MOVL C00062 V=800.0 PL=0
MOVL C00063 V=800.0 PL=0
MOVL C00064 V=800.0 PL=0
MOVL C00065 V=800.0 PL=0
MOVL C00066 V=800.0 PL=0
MOVL C00067 V=800.0 PL=0
MOVL C00068 V=800.0 PL=0
MOVL C00069 V=800.0 PL=0
MOVL C00070 V=800.0 PL=0
MOVL C00071 V=800.0 PL=0
MOVL C00072 V=800.0 PL=0
MOVL C00073 V=800.0 PL=0
MOVL C00074 V=800.0 PL=0
MOVL C00075 V=800.0 PL=0
MOVL C00076 V=800.0 PL=0
MOVL C00077 V=800.0 PL=0
MOVL C00078 V=800.0 PL=0
MOVL C00079 V=800.0 PL=0
MOVL C00080 V=800.0 PL=0
MOVL C00081 V=800.0 PL=0
MOVL C00082 V=800.0 PL=0
MOVL C00083 V=800.0 PL=0
MOVL C00084 V=800.0 PL=0
MOVL C00085 V=800.0 PL=0
MOVL C00086 V=800.0 PL=0
MOVL C00087 V=800.0 PL=0
MOVL C00088 V=800.0 PL=0
MOVL C00089 V=800.0 PL=0
MOVL C00090 V=800.0 PL=0
MOVL C00091 V=800.0 PL=0
MOVL C00092 V=800.0 PL=0
MOVL C00093 V=800.0 PL=0
MOVL C00094 V=800.0 PL=0
MOVL C00095 V=800.0 PL=0
MOVL C00096 V=800.0 PL=0
MOVL C00097 V=800.0 PL=0
MOVL C00098 V=800.0 PL=0
MOVL C00099 V=800.0 PL=0
MOVL C00100 V=800.0 PL=0
MOVL C00101 V=800.0 PL=0
MOVL C00102 V=800.0 PL=0
MOVL C00103 V=800.0 PL=0
MOVL C00104 V=800.0 PL=0
MOVL C00105 V=800.0 PL=0
MOVL C00106 V=800.0 PL=0
MOVL C00107 V=800.0 PL=0
MOVL C00108 V=800.0 PL=0
MOVL C00109 V=800.0 PL=0
MOVL C00110 V=800.0 PL=0
MOVL C00111 V=800.0 PL=0
MOVL C00112 V=800.0 PL=0
MOVL C00113 V=800.0 PL=0
MOVL C00114 V=800.0 PL=0
MOVL C00115 V=800.0 PL=0
MOVL C00116 V=800.0 PL=0
MOVL C00117 V=800.0 PL=0
MOVL C00118 V=800.0 PL=0
MOVL C00119 V=800.0 PL=0
MOVL C00120 V=800.0 PL=0
MOVL C00121 V=800.0 PL=0
MOVL C00122 V=800.0 PL=0
MOVL C00123 V=800.0 PL=0
MOVL C00124 V=800.0 PL=0
MOVL C00125 V=800.0 PL=0
MOVL C00126 V=800.0 PL=0
MOVL C00127 V=800.0 PL=0
MOVL C00128 V=800.0 PL=0
MOVL C00129 V=800.0 PL=0
MOVL C00130 V=800.0 PL=0
MOVL C00131 V=800.0 PL=0
MOVL C00132 V=800.0 PL=0
MOVL C00133 V=800.0 PL=0
MOVL C00134 V=800.0 PL=0
MOVL C00135 V=800.0 PL=0
MOVL C00136 V=800.0 PL=0
MOVL C00137 V=800.0 PL=0
MOVL C00138 V=800.0 PL=0
MOVL C00139 V=800.0 PL=0
MOVL C00140 V=800.0 PL=0
MOVL C00141 V=800.0 PL=0
MOVL C00142 V=800.0 PL=0
MOVL C00143 V=800.0 PL=0
MOVL C00144 V=800.0 PL=0
MOVL C00145 V=800.0 PL=0
MOVL C00146 V=800.0 PL=0
MOVL C00147 V=800.0 PL=0
MOVL C00148 V=800.0 PL=0
MOVL C00149 V=800.0 PL=0
MOVL C00150 V=800.0 PL=0
MOVL C00151 V=800.0 PL=0
MOVL C00152 V=800.0 PL=0
MOVL C00153 V=800.0 PL=0
MOVL C00154 V=800.0 PL=0
MOVL C00155 V=800.0 PL=0
MOVL C00156 V=800.0 PL=0
MOVL C00157 V=800.0 PL=0
MOVL C00158 V=800.0 PL=0
MOVL C00159 V=800.0 PL=0
MOVL C00160 V=800.0 PL=0
MOVL C00161 V=800.0 PL=0
MOVL C00162 V=800.0 PL=0
MOVL C00163 V=800.0 PL=0
MOVL C00164 V=800.0 PL=0
MOVL C00165 V=800.0 PL=0
MOVL C00166 V=800.0 PL=0
MOVL C00167 V=800.0 PL=0
MOVL C00168 V=800.0 PL=0
MOVL C00169 V=800.0 PL=0
MOVL C00170 V=800.0 PL=0
MOVL C00171 V=800.0 PL=0
MOVL C00172 V=800.0 PL=0
MOVL C00173 V=800.0 PL=0
MOVL C00174 V=800.0 PL=0
MOVL C00175 V=800.0 PL=0
MOVL C00176 V=800.0 PL=0
MOVL C00177 V=800.0 PL=0
MOVL C00178 V=800.0 PL=0
MOVL C00179 V=800.0 PL=0
MOVL C00180 V=800.0 PL=0
MOVL C00181 V=800.0 PL=0
MOVL C00182 V=800.0 PL=0
MOVL C00183 V=800.0 PL=0
MOVL C00184 V=800.0 PL=0
MOVL C00185 V=800.0 PL=0
MOVL C00186 V=800.0 PL=0
MOVL C00187 V=800.0 PL=0
MOVL C00188 V=800.0 PL=0
MOVL C00189 V=800.0 PL=0
MOVL C00190 V=800.0 PL=0
MOVL C00191 V=800.0 PL=0
MOVL C00192 V=800.0 PL=0
MOVL C00193 V=800.0 PL=0
MOVL C00194 V=800.0 PL=0
MOVL C00195 V=800.0 PL=0
MOVL C00196 V=800.0 PL=0
MOVL C00197 V=800.0 PL=0
MOVL C00198 V=800.0 PL=0
MOVL C00199 V=800.0 PL=0
MOVL C00200 V=800.0 PL=0
MOVL C00201 V=800.0 PL=0
MOVL C00202 V=800.0 PL=0
MOVL C00203 V=800.0 PL=0
MOVL C00204 V=800.0 PL=0
MOVL C00205 V=800.0 PL=0
MOVL C00206 V=800.0 PL=0
MOVL C00207 V=800.0 PL=0
MOVL C00208 V=800.0 PL=0
MOVL C00209 V=800.0 PL=0
MOVL C00210 V=800.0 PL=0
MOVL C00211 V=800.0 PL=0
MOVL C00212 V=800.0 PL=0
MOVL C00213 V=800.0 PL=0
MOVL C00214 V=800.0 PL=0
MOVL C00215 V=800.0 PL=0
MOVL C00216 V=800.0 PL=0
MOVL C00217 V=800.0 PL=0
MOVL C00218 V=800.0 PL=0
MOVL C00219 V=800.0 PL=0
MOVL C00220 V=800.0 PL=0
MOVL C00221 V=800.0 PL=0
MOVL C00222 V=800.0 PL=0
MOVL C00223 V=800.0 PL=0
MOVL C00224 V=800.0 PL=0
MOVL C00225 V=800.0 PL=0
MOVL C00226 V=800.0 PL=0
MOVL C00227 V=800.0 PL=0
MOVL C00228 V=800.0 PL=0
MOVL C00229 V=800.0 PL=0
MOVL C00230 V=800.0 PL=0
MOVL C00231 V=800.0 PL=0
MOVL C00232 V=800.0 PL=0
MOVL C00233 V=800.0 PL=0
MOVL C00234 V=800.0 PL=0
MOVL C00235 V=800.0 PL=0
MOVL C00236 V=800.0 PL=0
MOVL C00237 V=800.0 PL=0
MOVL C00238 V=800.0 PL=0
MOVL C00239 V=800.0 PL=0
MOVL C00240 V=800.0 PL=0
MOVL C00241 V=800.0 PL=0
MOVL C00242 V=800.0 PL=0
MOVL C00243 V=800.0 PL=0
MOVL C00244 V=800.0 PL=0
MOVL C00245 V=800.0 PL=0
MOVL C00246 V=800.0 PL=0
MOVL C00247 V=800.0 PL=0
MOVL C00248 V=800.0 PL=0
MOVL C00249 V=800.0 PL=0
MOVL C00250 V=800.0 PL=0
MOVL C00251 V=800.0 PL=0
MOVL C00252 V=800.0 PL=0
MOVL C00253 V=800.0 PL=0
MOVL C00254 V=800.0 PL=0
MOVL C00255 V=800.0 PL=0
MOVL C00256 V=800.0 PL=0
MOVL C00257 V=800.0 PL=0
MOVL C00258 V=800.0 PL=0
MOVL C00259 V=800.0 PL=0
MOVL C00260 V=800.0 PL=0
MOVL C00261 V=800.0 PL=0
MOVL C00262 V=800.0 PL=0
MOVL C00263 V=800.0 PL=0
MOVL C00264 V=800.0 PL=0
MOVL C00265 V=800.0 PL=0
MOVL C00266 V=800.0 PL=0
MOVL C00267 V=800.0 PL=0
MOVL C00268 V=800.0 PL=0
MOVL C00269 V=800.0 PL=0
MOVL C00270 V=800.0 PL=0
MOVL C00271 V=800.0 PL=0
MOVL C00272 V=800.0 PL=0
MOVL C00273 V=800.0 PL=0
MOVL C00274 V=800.0 PL=0
MOVL C00275 V=800.0 PL=0
MOVL C00276 V=800.0 PL=0
MOVL C00277 V=800.0 PL=0
MOVL C00278 V=800.0 PL=0
MOVL C00279 V=800.0 PL=0
MOVL C00280 V=800.0 PL=0
MOVL C00281 V=800.0 PL=0
MOVL C00282 V=800.0 PL=0
MOVL C00283 V=800.0 PL=0
MOVL C00284 V=800.0 PL=0
MOVL C00285 V=800.0 PL=0
MOVL C00286 V=800.0 PL=0
MOVL C00287 V=800.0 PL=0
MOVL C00288 V=800.0 PL=0
MOVL C00289 V=800.0 PL=0
MOVL C00290 V=800.0 PL=0
MOVL C00291 V=800.0 PL=0
MOVL C00292 V=800.0 PL=0
MOVL C00293 V=800.0 PL=0
MOVL C00294 V=800.0 PL=0
MOVL C00295 V=800.0 PL=0
MOVL C00296 V=800.0 PL=0
MOVL C00297 V=800.0 PL=0
MOVL C00298 V=800.0 PL=0
MOVL C00299 V=800.0 PL=0
MOVL C00300 V=800.0 PL=0
MOVL C00301 V=800.0 PL=0
MOVL C00302 V=800.0 PL=0
MOVL C00303 V=800.0 PL=0
MOVL C00304 V=800.0 PL=0
MOVL C00305 V=800.0 PL=0
MOVL C00306 V=800.0 PL=0
MOVL C00307 V=800.0 PL=0
MOVL C00308 V=800.0 PL=0
MOVL C00309 V=800.0 PL=0
MOVL C00310 V=800.0 PL=0
MOVL C00311 V=800.0 PL=0
MOVL C00312 V=800.0 PL=0
MOVL C00313 V=800.0 PL=0
MOVL C00314 V=800.0 PL=0
MOVL C00315 V=800.0 PL=0
MOVL C00316 V=800.0 PL=0
MOVL C00317 V=800.0 PL=0
MOVL C00318 V=800.0 PL=0
MOVL C00319 V=800.0 PL=0
MOVL C00320 V=800.0 PL=0
MOVL C00321 V=800.0 PL=0
MOVL C00322 V=800.0 PL=0
MOVL C00323 V=800.0 PL=0
MOVL C00324 V=800.0 PL=0
MOVL C00325 V=800.0 PL=0
MOVL C00326 V=800.0 PL=0
MOVL C00327 V=800.0 PL=0
MOVL C00328 V=800.0 PL=0
MOVL C00329 V=800.0 PL=0
MOVL C00330 V=800.0 PL=0
MOVL C00331 V=800.0 PL=0
MOVL C00332 V=800.0 PL=0
MOVL C00333 V=800.0 PL=0
MOVL C00334 V=800.0 PL=0
MOVL C00335 V=800.0 PL=0
MOVL C00336 V=800.0 PL=0
MOVL C00337 V=800.0 PL=0
MOVL C00338 V=800.0 PL=0
MOVL C00339 V=800.0 PL=0
MOVL C00340 V=800.0 PL=0
MOVL C00341 V=800.0 PL=0
MOVL C00342 V=800.0 PL=0
MOVL C00343 V=800.0 PL=0
MOVL C00344 V=800.0 PL=0
MOVL C00345 V=800.0 PL=0
MOVL C00346 V=800.0 PL=0
MOVL C00347 V=800.0 PL=0
MOVL C00348 V=800.0 PL=0
MOVL C00349 V=800.0 PL=0
MOVL C00350 V=800.0 PL=0
MOVL C00351 V=800.0 PL=0
MOVL C00352 V=800.0 PL=0
MOVL C00353 V=800.0 PL=0
MOVL C00354 V=800.0 PL=0
MOVL C00355 V=800.0 PL=0
MOVL C00356 V=800.0 PL=0
MOVL C00357 V=800.0 PL=0
MOVL C00358 V=800.0 PL=0
MOVL C00359 V=800.0 PL=0
MOVL C00360 V=800.0 PL=0
MOVL C00361 V=800.0 PL=0
MOVL C00362 V=800.0 PL=0
MOVL C00363 V=800.0 PL=0
MOVL C00364 V=800.0 PL=0
MOVL C00365 V=800.0 PL=0
MOVL C00366 V=800.0 PL=0
MOVL C00367 V=800.0 PL=0
MOVL C00368 V=800.0 PL=0
MOVL C00369 V=800.0 PL=0
MOVL C00370 V=800.0 PL=0
MOVL C00371 V=800.0 PL=0
MOVL C00372 V=800.0 PL=0
MOVL C00373 V=800.0 PL=0
MOVL C00374 V=800.0 PL=0
MOVL C00375 V=800.0 PL=0
MOVL C00376 V=800.0 PL=0
MOVL C00377 V=800.0 PL=0
MOVL C00378 V=800.0 PL=0
MOVL C00379 V=800.0 PL=0
MOVL C00380 V=800.0 PL=0
MOVL C00381 V=800.0 PL=0
MOVL C00382 V=800.0 PL=0
MOVL C00383 V=800.0 PL=0
MOVL C00384 V=800.0 PL=0
MOVL C00385 V=800.0 PL=0
MOVL C00386 V=800.0 PL=0
MOVL C00387 V=800.0 PL=0
MOVL C00388 V=800.0 PL=0
MOVL C00389 V=800.0 PL=0
MOVL C00390 V=800.0 PL=0
MOVL C00391 V=800.0 PL=0
MOVL C00392 V=800.0 PL=0
MOVL C00393 V=800.0 PL=0
MOVL C00394 V=800.0 PL=0
MOVL C00395 V=800.0 PL=0
MOVL C00396 V=800.0 PL=0
MOVL C00397 V=800.0 PL=0
MOVL C00398 V=800.0 PL=0
MOVL C00399 V=800.0 PL=0
MOVL C00400 V=800.0 PL=0
MOVL C00401 V=800.0 PL=0
MOVL C00402 V=800.0 PL=0
MOVL C00403 V=800.0 PL=0
MOVL C00404 V=800.0 PL=0
MOVL C00405 V=800.0 PL=0
MOVL C00406 V=800.0 PL=0
MOVL C00407 V=800.0 PL=0
MOVL C00408 V=800.0 PL=0
MOVL C00409 V=800.0 PL=0
MOVL C00410 V=800.0 PL=0
MOVL C00411 V=800.0 PL=0
MOVL C00412 V=800.0 PL=0
MOVL C00413 V=800.0 PL=0
MOVL C00414 V=800.0 PL=0
MOVL C00415 V=800.0 PL=0
MOVL C00416 V=800.0 PL=0
MOVL C00417 V=800.0 PL=0
MOVL C00418 V=800.0 PL=0
MOVL C00419 V=800.0 PL=0
MOVL C00420 V=800.0 PL=0
MOVL C00421 V=800.0 PL=0
MOVL C00422 V=800.0 PL=0
MOVL C00423 V=800.0 PL=0
MOVL C00424 V=800.0 PL=0
MOVL C00425 V=800.0 PL=0
MOVL C00426 V=800.0 PL=0
MOVL C00427 V=800.0 PL=0
MOVL C00428 V=800.0 PL=0
MOVL C00429 V=800.0 PL=0
MOVL C00430 V=800.0 PL=0
MOVL C00431 V=800.0 PL=0
MOVL C00432 V=800.0 PL=0
MOVL C00433 V=800.0 PL=0
MOVL C00434 V=800.0 PL=0
MOVL C00435 V=800.0 PL=0
MOVL C00436 V=800.0 PL=0
MOVL C00437 V=800.0 PL=0
MOVL C00438 V=800.0 PL=0
MOVL C00439 V=800.0 PL=0
MOVL C00440 V=800.0 PL=0
MOVL C00441 V=800.0 PL=0
MOVL C00442 V=800.0 PL=0
MOVL C00443 V=800.0 PL=0
MOVL C00444 V=800.0 PL=0
MOVL C00445 V=800.0 PL=0
MOVL C00446 V=800.0 PL=0
MOVL C00447 V=800.0 PL=0
MOVL C00448 V=800.0 PL=0
MOVL C00449 V=800.0 PL=0
MOVL C00450 V=800.0 PL=0
MOVL C00451 V=800.0 PL=0
MOVL C00452 V=800.0 PL=0
MOVL C00453 V=800.0 PL=0
MOVL C00454 V=800.0 PL=0
MOVL C00455 V=800.0 PL=0
MOVL C00456 V=800.0 PL=0
MOVL C00457 V=800.0 PL=0
MOVL C00458 V=800.0 PL=0
MOVL C00459 V=800.0 PL=0
MOVL C00460 V=800.0 PL=0
MOVL C00461 V=800.0 PL=0
MOVL C00462 V=800.0 PL=0
MOVL C00463 V=800.0 PL=0
MOVL C00464 V=800.0 PL=0
MOVL C00465 V=800.0 PL=0
MOVL C00466 V=800.0 PL=0
MOVL C00467 V=800.0 PL=0
MOVL C00468 V=800.0 PL=0
MOVL C00469 V=800.0 PL=0
MOVL C00470 V=800.0 PL=0
MOVL C00471 V=800.0 PL=0
MOVL C00472 V=800.0 PL=0
MOVL C00473 V=800.0 PL=0
MOVL C00474 V=800.0 PL=0
MOVL C00475 V=800.0 PL=0
MOVL C00476 V=800.0 PL=0
MOVL C00477 V=800.0 PL=0
MOVL C00478 V=800.0 PL=0
MOVL C00479 V=800.0 PL=0
MOVL C00480 V=800.0 PL=0
MOVL C00481 V=800.0 PL=0
MOVL C00482 V=800.0 PL=0
MOVL C00483 V=800.0 PL=0
MOVL C00484 V=800.0 PL=0
MOVL C00485 V=800.0 PL=0
MOVL C00486 V=800.0 PL=0
MOVL C00487 V=800.0 PL=0
MOVL C00488 V=800.0 PL=0
MOVL C00489 V=800.0 PL=0
MOVL C00490 V=800.0 PL=0
MOVL C00491 V=800.0 PL=0
MOVL C00492 V=800.0 PL=0
MOVL C00493 V=800.0 PL=0
MOVL C00494 V=800.0 PL=0
MOVL C00495 V=800.0 PL=0
MOVL C00496 V=800.0 PL=0
MOVL C00497 V=800.0 PL=0
MOVL C00498 V=800.0 PL=0
MOVL C00499 V=800.0 PL=0
MOVL C00500 V=800.0 PL=0
MOVL C00501 V=800.0 PL=0
MOVL C00502 V=800.0 PL=0
MOVL C00503 V=800.0 PL=0
MOVL C00504 V=800.0 PL=0
MOVL C00505 V=800.0 PL=0
MOVL C00506 V=800.0 PL=0
MOVL C00507 V=800.0 PL=0
MOVL C00508 V=800.0 PL=0
MOVL C00509 V=800.0 PL=0
MOVL C00510 V=800.0 PL=0
MOVL C00511 V=800.0 PL=0
MOVL C00512 V=800.0 PL=0
MOVL C00513 V=800.0 PL=0
MOVL C00514 V=800.0 PL=0
MOVL C00515 V=800.0 PL=0
MOVL C00516 V=800.0 PL=0
MOVL C00517 V=800.0 PL=0
MOVL C00518 V=800.0 PL=0
MOVL C00519 V=800.0 PL=0
MOVL C00520 V=800.0 PL=0
MOVL C00521 V=800.0 PL=0
MOVL C00522 V=800.0 PL=0
MOVL C00523 V=800.0 PL=0
MOVL C00524 V=800.0 PL=0
MOVL C00525 V=800.0 PL=0
MOVL C00526 V=800.0 PL=0
MOVL C00527 V=800.0 PL=0
MOVL C00528 V=800.0 PL=0
MOVL C00529 V=800.0 PL=0
MOVL C00530 V=800.0 PL=0
MOVL C00531 V=800.0 PL=0
MOVL C00532 V=800.0 PL=0
MOVL C00533 V=800.0 PL=0
MOVL C00534 V=800.0 PL=0
MOVL C00535 V=800.0 PL=0
MOVL C00536 V=800.0 PL=0
MOVL C00537 V=800.0 PL=0
MOVL C00538 V=800.0 PL=0
MOVL C00539 V=800.0 PL=0
MOVL C00540 V=800.0 PL=0
MOVL C00541 V=800.0 PL=0
MOVL C00542 V=800.0 PL=0
MOVL C00543 V=800.0 PL=0
MOVL C00544 V=800.0 PL=0
MOVL C00545 V=800.0 PL=0
MOVL C00546 V=800.0 PL=0
MOVL C00547 V=800.0 PL=0
MOVL C00548 V=800.0 PL=0
MOVL C00549 V=800.0 PL=0
MOVL C00550 V=800.0 PL=0
MOVL C00551 V=800.0 PL=0
MOVL C00552 V=800.0 PL=0
MOVL C00553 V=800.0 PL=0
MOVL C00554 V=800.0 PL=0
MOVL C00555 V=800.0 PL=0
MOVL C00556 V=800.0 PL=0
MOVL C00557 V=800.0 PL=0
MOVL C00558 V=800.0 PL=0
MOVL C00559 V=800.0 PL=0
MOVL C00560 V=800.0 PL=0
MOVL C00561 V=800.0 PL=0
MOVL C00562 V=800.0 PL=0
MOVL C00563 V=800.0 PL=0
MOVL C00564 V=800.0 PL=0
MOVL C00565 V=800.0 PL=0
MOVL C00566 V=800.0 PL=0
MOVL C00567 V=800.0 PL=0
MOVL C00568 V=800.0 PL=0
MOVL C00569 V=800.0 PL=0
MOVL C00570 V=800.0 PL=0
MOVL C00571 V=800.0 PL=0
MOVL C00572 V=800.0 PL=0
MOVL C00573 V=800.0 PL=0
MOVL C00574 V=800.0 PL=0
MOVL C00575 V=800.0 PL=0
MOVL C00576 V=800.0 PL=0
MOVL C00577 V=800.0 PL=0
MOVL C00578 V=800.0 PL=0
MOVL C00579 V=800.0 PL=0
MOVL C00580 V=800.0 PL=0
MOVL C00581 V=800.0 PL=0
MOVL C00582 V=800.0 PL=0
MOVL C00583 V=800.0 PL=0
MOVL C00584 V=800.0 PL=0
MOVL C00585 V=800.0 PL=0
MOVL C00586 V=800.0 PL=0
MOVL C00587 V=800.0 PL=0
MOVL C00588 V=800.0 PL=0
MOVL C00589 V=800.0 PL=0
MOVL C00590 V=800.0 PL=0
MOVL C00591 V=800.0 PL=0
MOVL C00592 V=800.0 PL=0
MOVL C00593 V=800.0 PL=0
MOVL C00594 V=800.0 PL=0
MOVL C00595 V=800.0 PL=0
MOVL C00596 V=800.0 PL=0
MOVL C00597 V=800.0 PL=0
MOVL C00598 V=800.0 PL=0
MOVL C00599 V=800.0 PL=0
MOVL C00600 V=800.0 PL=0
MOVL C00601 V=800.0 PL=0
MOVL C00602 V=800.0 PL=0
MOVL C00603 V=800.0 PL=0
MOVL C00604 V=800.0 PL=0
MOVL C00605 V=800.0 PL=0
MOVL C00606 V=800.0 PL=0
MOVL C00607 V=800.0 PL=0
MOVL C00608 V=800.0 PL=0
MOVL C00609 V=800.0 PL=0
MOVL C00610 V=800.0 PL=0
MOVL C00611 V=800.0 PL=0
MOVL C00612 V=800.0 PL=0
MOVL C00613 V=800.0 PL=0
MOVL C00614 V=800.0 PL=0
MOVL C00615 V=800.0 PL=0
MOVL C00616 V=800.0 PL=0
MOVL C00617 V=800.0 PL=0
MOVL C00618 V=800.0 PL=0
MOVL C00619 V=800.0 PL=0
MOVL C00620 V=800.0 PL=0
MOVL C00621 V=800.0 PL=0
MOVL C00622 V=800.0 PL=0
MOVL C00623 V=800.0 PL=0
MOVL C00624 V=800.0 PL=0
MOVL C00625 V=800.0 PL=0
MOVL C00626 V=800.0 PL=0
MOVL C00627 V=800.0 PL=0
MOVL C00628 V=800.0 PL=0
MOVL C00629 V=800.0 PL=0
MOVL C00630 V=800.0 PL=0
MOVL C00631 V=800.0 PL=0
MOVL C00632 V=800.0 PL=0
MOVL C00633 V=800.0 PL=0
MOVL C00634 V=800.0 PL=0
MOVL C00635 V=800.0 PL=0
MOVL C00636 V=800.0 PL=0
MOVL C00637 V=800.0 PL=0
MOVL C00638 V=800.0 PL=0
MOVL C00639 V=800.0 PL=0
MOVL C00640 V=800.0 PL=0
MOVL C00641 V=800.0 PL=0
MOVL C00642 V=800.0 PL=0
MOVL C00643 V=800.0 PL=0
MOVL C00644 V=800.0 PL=0
MOVL C00645 V=800.0 PL=0
MOVL C00646 V=800.0 PL=0
MOVL C00647 V=800.0 PL=0
MOVL C00648 V=800.0 PL=0
MOVL C00649 V=800.0 PL=0
MOVL C00650 V=800.0 PL=0
MOVL C00651 V=800.0 PL=0
MOVL C00652 V=800.0 PL=0
MOVL C00653 V=800.0 PL=0
MOVL C00654 V=800.0 PL=0
MOVL C00655 V=800.0 PL=0
MOVL C00656 V=800.0 PL=0
MOVL C00657 V=800.0 PL=0
MOVL C00658 V=800.0 PL=0
MOVL C00659 V=800.0 PL=0
MOVL C00660 V=800.0 PL=0
MOVL C00661 V=800.0 PL=0
MOVL C00662 V=800.0 PL=0
MOVL C00663 V=800.0 PL=0
MOVL C00664 V=800.0 PL=0
MOVL C00665 V=800.0 PL=0
MOVL C00666 V=800.0 PL=0
MOVL C00667 V=800.0 PL=0
MOVL C00668 V=800.0 PL=0
MOVL C00669 V=800.0 PL=0
MOVL C00670 V=800.0 PL=0
MOVL C00671 V=800.0 PL=0
MOVL C00672 V=800.0 PL=0
MOVL C00673 V=800.0 PL=0
MOVL C00674 V=800.0 PL=0
MOVL C00675 V=800.0 PL=0
MOVL C00676 V=800.0 PL=0
MOVL C00677 V=800.0 PL=0
MOVL C00678 V=800.0 PL=0
MOVL C00679 V=800.0 PL=0
MOVL C00680 V=800.0 PL=0
MOVL C00681 V=800.0 PL=0
MOVL C00682 V=800.0 PL=0
MOVL C00683 V=800.0 PL=0
MOVL C00684 V=800.0 PL=0
MOVL C00685 V=800.0 PL=0
MOVL C00686 V=800.0 PL=0
MOVL C00687 V=800.0 PL=0
MOVL C00688 V=800.0 PL=0
MOVL C00689 V=800.0 PL=0
MOVL C00690 V=800.0 PL=0
MOVL C00691 V=800.0 PL=0
MOVL C00692 V=800.0 PL=0
MOVL C00693 V=800.0 PL=0
MOVL C00694 V=800.0 PL=0
MOVL C00695 V=800.0 PL=0
MOVL C00696 V=800.0 PL=0
MOVL C00697 V=800.0 PL=0
MOVL C00698 V=800.0 PL=0
MOVL C00699 V=800.0 PL=0
MOVL C00700 V=800.0 PL=0
MOVL C00701 V=800.0 PL=0
MOVL C00702 V=800.0 PL=0
MOVL C00703 V=800.0 PL=0
MOVL C00704 V=800.0 PL=0
MOVL C00705 V=800.0 PL=0
MOVL C00706 V=800.0 PL=0
MOVL C00707 V=800.0 PL=0
MOVL C00708 V=800.0 PL=0
MOVL C00709 V=800.0 PL=0
MOVL C00710 V=800.0 PL=0
MOVL C00711 V=800.0 PL=0
MOVL C00712 V=800.0 PL=0
MOVL C00713 V=800.0 PL=0
MOVL C00714 V=800.0 PL=0
MOVL C00715 V=800.0 PL=0
MOVL C00716 V=800.0 PL=0
MOVL C00717 V=800.0 PL=0
MOVL C00718 V=800.0 PL=0
MOVL C00719 V=800.0 PL=0
MOVL C00720 V=800.0 PL=0
MOVL C00721 V=800.0 PL=0
MOVL C00722 V=800.0 PL=0
MOVL C00723 V=800.0 PL=0
MOVL C00724 V=800.0 PL=0
MOVL C00725 V=800.0 PL=0
MOVL C00726 V=800.0 PL=0
MOVL C00727 V=800.0 PL=0
MOVL C00728 V=800.0 PL=0
MOVL C00729 V=800.0 PL=0
MOVL C00730 V=800.0 PL=0
MOVL C00731 V=800.0 PL=0
MOVL C00732 V=800.0 PL=0
MOVL C00733 V=800.0 PL=0
MOVL C00734 V=800.0 PL=0
MOVL C00735 V=800.0 PL=0
MOVL C00736 V=800.0 PL=0
MOVL C00737 V=800.0 PL=0
MOVL C00738 V=800.0 PL=0
MOVL C00739 V=800.0 PL=0
MOVL C00740 V=800.0 PL=0
MOVL C00741 V=800.0 PL=0
MOVL C00742 V=800.0 PL=0
MOVL C00743 V=800.0 PL=0
MOVL C00744 V=800.0 PL=0
MOVL C00745 V=800.0 PL=0
MOVL C00746 V=800.0 PL=0
MOVL C00747 V=800.0 PL=0
MOVL C00748 V=800.0 PL=0
MOVL C00749 V=800.0 PL=0
MOVL C00750 V=800.0 PL=0
MOVL C00751 V=800.0 PL=0
MOVL C00752 V=800.0 PL=0
MOVL C00753 V=800.0 PL=0
MOVL C00754 V=800.0 PL=0
MOVL C00755 V=800.0 PL=0
MOVL C00756 V=800.0 PL=0
MOVL C00757 V=800.0 PL=0
MOVL C00758 V=800.0 PL=0
MOVL C00759 V=800.0 PL=0
MOVL C00760 V=800.0 PL=0
MOVL C00761 V=800.0 PL=0
MOVL C00762 V=800.0 PL=0
MOVL C00763 V=800.0 PL=0
MOVL C00764 V=800.0 PL=0
MOVL C00765 V=800.0 PL=0
MOVL C00766 V=800.0 PL=0
MOVL C00767 V=800.0 PL=0
MOVL C00768 V=800.0 PL=0
MOVL C00769 V=800.0 PL=0
MOVL C00770 V=800.0 PL=0
MOVL C00771 V=800.0 PL=0
MOVL C00772 V=800.0 PL=0
MOVL C00773 V=800.0 PL=0
MOVL C00774 V=800.0 PL=0
MOVL C00775 V=800.0 PL=0
MOVL C00776 V=800.0 PL=0
MOVL C00777 V=800.0 PL=0
MOVL C00778 V=800.0 PL=0
MOVL C00779 V=800.0 PL=0
MOVL C00780 V=800.0 PL=0
MOVL C00781 V=800.0 PL=0
MOVL C00782 V=800.0 PL=0
MOVL C00783 V=800.0 PL=0
MOVL C00784 V=800.0 PL=0
MOVL C00785 V=800.0 PL=0
MOVL C00786 V=800.0 PL=0
MOVL C00787 V=800.0 PL=0
MOVL C00788 V=800.0 PL=0
MOVL C00789 V=800.0 PL=0
MOVL C00790 V=800.0 PL=0
MOVL C00791 V=800.0 PL=0
MOVL C00792 V=800.0 PL=0
MOVL C00793 V=800.0 PL=0
MOVL C00794 V=800.0 PL=0
MOVL C00795 V=800.0 PL=0
MOVL C00796 V=800.0 PL=0
MOVL C00797 V=800.0 PL=0
MOVL C00798 V=800.0 PL=0
MOVL C00799 V=800.0 PL=0
MOVL C00800 V=800.0 PL=0
MOVL C00801 V=800.0 PL=0
MOVL C00802 V=800.0 PL=0
MOVL C00803 V=800.0 PL=0
MOVL C00804 V=800.0 PL=0
MOVL C00805 V=800.0 PL=0
MOVL C00806 V=800.0 PL=0
MOVL C00807 V=800.0 PL=0
MOVL C00808 V=800.0 PL=0
MOVL C00809 V=800.0 PL=0
MOVL C00810 V=800.0 PL=0
MOVL C00811 V=800.0 PL=0
MOVL C00812 V=800.0 PL=0
MOVL C00813 V=800.0 PL=0
MOVL C00814 V=800.0 PL=0
MOVL C00815 V=800.0 PL=0
MOVL C00816 V=800.0 PL=0
MOVL C00817 V=800.0 PL=0
MOVL C00818 V=800.0 PL=0
MOVL C00819 V=800.0 PL=0
MOVL C00820 V=800.0 PL=0
MOVL C00821 V=800.0 PL=0
MOVL C00822 V=800.0 PL=0
MOVL C00823 V=800.0 PL=0
MOVL C00824 V=800.0 PL=0
MOVL C00825 V=800.0 PL=0
MOVL C00826 V=800.0 PL=0
MOVL C00827 V=800.0 PL=0
MOVL C00828 V=800.0 PL=0
MOVL C00829 V=800.0 PL=0
MOVL C00830 V=800.0 PL=0
MOVL C00831 V=800.0 PL=0
MOVL C00832 V=800.0 PL=0
MOVL C00833 V=800.0 PL=0
MOVL C00834 V=800.0 PL=0
MOVL C00835 V=800.0 PL=0
MOVL C00836 V=800.0 PL=0
MOVL C00837 V=800.0 PL=0
MOVL C00838 V=800.0 PL=0
MOVL C00839 V=800.0 PL=0
MOVL C00840 V=800.0 PL=0
MOVL C00841 V=800.0 PL=0
MOVL C00842 V=800.0 PL=0
MOVL C00843 V=800.0 PL=0
MOVL C00844 V=800.0 PL=0
MOVL C00845 V=800.0 PL=0
MOVL C00846 V=800.0 PL=0
MOVL C00847 V=800.0 PL=0
MOVL C00848 V=800.0 PL=0
MOVL C00849 V=800.0 PL=0
MOVL C00850 V=800.0 PL=0
MOVL C00851 V=800.0 PL=0
MOVL C00852 V=800.0 PL=0
MOVL C00853 V=800.0 PL=0
MOVL C00854 V=800.0 PL=0
MOVL C00855 V=800.0 PL=0
MOVL C00856 V=800.0 PL=0
MOVL C00857 V=800.0 PL=0
MOVL C00858 V=800.0 PL=0
MOVL C00859 V=800.0 PL=0
MOVL C00860 V=800.0 PL=0
MOVL C00861 V=800.0 PL=0
MOVL C00862 V=800.0 PL=0
MOVL C00863 V=800.0 PL=0
MOVL C00864 V=800.0 PL=0
MOVL C00865 V=800.0 PL=0
MOVL C00866 V=800.0 PL=0
MOVL C00867 V=800.0 PL=0
MOVL C00868 V=800.0 PL=0
MOVL C00869 V=800.0 PL=0
MOVL C00870 V=800.0 PL=0
MOVL C00871 V=800.0 PL=0
MOVL C00872 V=800.0 PL=0
MOVL C00873 V=800.0 PL=0
MOVL C00874 V=800.0 PL=0
MOVL C00875 V=800.0 PL=0
MOVL C00876 V=800.0 PL=0
MOVL C00877 V=800.0 PL=0
MOVL C00878 V=800.0 PL=0
MOVL C00879 V=800.0 PL=0
MOVL C00880 V=800.0 PL=0
MOVL C00881 V=800.0 PL=0
MOVL C00882 V=800.0 PL=0
MOVL C00883 V=800.0 PL=0
MOVL C00884 V=800.0 PL=0
MOVL C00885 V=800.0 PL=0
MOVL C00886 V=800.0 PL=0
MOVL C00887 V=800.0 PL=0
MOVL C00888 V=800.0 PL=0
MOVL C00889 V=800.0 PL=0
MOVL C00890 V=800.0 PL=0
MOVL C00891 V=800.0 PL=0
MOVL C00892 V=800.0 PL=0
MOVL C00893 V=800.0 PL=0
MOVL C00894 V=800.0 PL=0
MOVL C00895 V=800.0 PL=0
MOVL C00896 V=800.0 PL=0
MOVL C00897 V=800.0 PL=0
MOVL C00898 V=800.0 PL=0
MOVL C00899 V=800.0 PL=0
MOVL C00900 V=800.0 PL=0
MOVL C00901 V=800.0 PL=0
MOVL C00902 V=800.0 PL=0
MOVL C00903 V=800.0 PL=0
MOVL C00904 V=800.0 PL=0
MOVL C00905 V=800.0 PL=0
MOVL C00906 V=800.0 PL=0
MOVL C00907 V=800.0 PL=0
MOVL C00908 V=800.0 PL=0
MOVL C00909 V=800.0 PL=0
MOVL C00910 V=800.0 PL=0
MOVL C00911 V=800.0 PL=0
MOVL C00912 V=800.0 PL=0
MOVL C00913 V=800.0 PL=0
MOVL C00914 V=800.0 PL=0
MOVL C00915 V=800.0 PL=0
MOVL C00916 V=800.0 PL=0
MOVL C00917 V=800.0 PL=0
MOVL C00918 V=800.0 PL=0
MOVL C00919 V=800.0 PL=0
MOVL C00920 V=800.0 PL=0
MOVL C00921 V=800.0 PL=0
MOVL C00922 V=800.0 PL=0
MOVL C00923 V=800.0 PL=0
MOVL C00924 V=800.0 PL=0
MOVL C00925 V=800.0 PL=0
MOVL C00926 V=800.0 PL=0
MOVL C00927 V=800.0 PL=0
MOVL C00928 V=800.0 PL=0
MOVL C00929 V=800.0 PL=0
MOVL C00930 V=800.0 PL=0
MOVL C00931 V=800.0 PL=0
MOVL C00932 V=800.0 PL=0
MOVL C00933 V=800.0 PL=0
MOVL C00934 V=800.0 PL=0
MOVL C00935 V=800.0 PL=0
MOVL C00936 V=800.0 PL=0
MOVL C00937 V=800.0 PL=0
MOVL C00938 V=800.0 PL=0
MOVL C00939 V=800.0 PL=0
MOVL C00940 V=800.0 PL=0
MOVL C00941 V=800.0 PL=0
MOVL C00942 V=800.0 PL=0
MOVL C00943 V=800.0 PL=0
MOVL C00944 V=800.0 PL=0
MOVL C00945 V=800.0 PL=0
MOVL C00946 V=800.0 PL=0
MOVL C00947 V=800.0 PL=0
MOVL C00948 V=800.0 PL=0
MOVL C00949 V=800.0 PL=0
MOVL C00950 V=800.0 PL=0
MOVL C00951 V=800.0 PL=0
MOVL C00952 V=800.0 PL=0
MOVL C00953 V=800.0 PL=0
MOVL C00954 V=800.0 PL=0
MOVL C00955 V=800.0 PL=0
MOVL C00956 V=800.0 PL=0
MOVL C00957 V=800.0 PL=0
MOVL C00958 V=800.0 PL=0
MOVL C00959 V=800.0 PL=0
MOVL C00960 V=800.0 PL=0
MOVL C00961 V=800.0 PL=0
MOVL C00962 V=800.0 PL=0
MOVL C00963 V=800.0 PL=0
MOVL C00964 V=800.0 PL=0
MOVL C00965 V=800.0 PL=0
MOVL C00966 V=800.0 PL=0
MOVL C00967 V=800.0 PL=0
MOVL C00968 V=800.0 PL=0
MOVL C00969 V=800.0 PL=0
MOVL C00970 V=800.0 PL=0
MOVL C00971 V=800.0 PL=0
MOVL C00972 V=800.0 PL=0
MOVL C00973 V=800.0 PL=0
MOVL C00974 V=800.0 PL=0
MOVL C00975 V=800.0 PL=0
MOVL C00976 V=800.0 PL=0
MOVL C00977 V=800.0 PL=0
MOVL C00978 V=800.0 PL=0
MOVL C00979 V=800.0 PL=0
MOVL C00980 V=800.0 PL=0
MOVL C00981 V=800.0 PL=0
MOVL C00982 V=800.0 PL=0
MOVL C00983 V=800.0 PL=0
MOVL C00984 V=800.0 PL=0
MOVL C00985 V=800.0 PL=0
MOVL C00986 V=800.0 PL=0
MOVL C00987 V=800.0 PL=0
MOVL C00988 V=800.0 PL=0
MOVL C00989 V=800.0 PL=0
MOVL C00990 V=800.0 PL=0
MOVL C00991 V=800.0 PL=0
MOVL C00992 V=800.0 PL=0
MOVL C00993 V=800.0 PL=0
MOVL C00994 V=800.0 PL=0
MOVL C00995 V=800.0 PL=0
MOVL C00996 V=800.0 PL=0
MOVL C00997 V=800.0 PL=0
MOVL C00998 V=800.0 PL=0
MOVL C00999 V=800.0 PL=0
MOVL C01000 V=800.0 PL=0
MOVL C01001 V=800.0 PL=0
MOVL C01002 V=800.0 PL=0
MOVL C01003 V=800.0 PL=0
MOVL C01004 V=800.0 PL=0
MOVL C01005 V=800.0 PL=0
MOVL C01006 V=800.0 PL=0
MOVL C01007 V=800.0 PL=0
MOVL C01008 V=800.0 PL=0
MOVL C01009 V=800.0 PL=0
MOVL C01010 V=800.0 PL=0
MOVL C01011 V=800.0 PL=0
MOVL C01012 V=800.0 PL=0
MOVL C01013 V=800.0 PL=0
MOVL C01014 V=800.0 PL=0
MOVL C01015 V=800.0 PL=0
MOVL C01016 V=800.0 PL=0
MOVL C01017 V=800.0 PL=0
MOVL C01018 V=800.0 PL=0
MOVL C01019 V=800.0 PL=0
MOVL C01020 V=800.0 PL=0
MOVL C01021 V=800.0 PL=0
MOVL C01022 V=800.0 PL=0
MOVL C01023 V=800.0 PL=0
MOVL C01024 V=800.0 PL=0
MOVL C01025 V=800.0 PL=0
MOVL C01026 V=800.0 PL=0
MOVL C01027 V=800.0 PL=0
MOVL C01028 V=800.0 PL=0
MOVL C01029 V=800.0 PL=0
MOVL C01030 V=800.0 PL=0
MOVL C01031 V=800.0 PL=0
MOVL C01032 V=800.0 PL=0
MOVL C01033 V=800.0 PL=0
MOVL C01034 V=800.0 PL=0
MOVL C01035 V=800.0 PL=0
MOVL C01036 V=800.0 PL=0
MOVL C01037 V=800.0 PL=0
MOVL C01038 V=800.0 PL=0
MOVL C01039 V=800.0 PL=0
MOVL C01040 V=800.0 PL=0
MOVL C01041 V=800.0 PL=0
MOVL C01042 V=800.0 PL=0
MOVL C01043 V=800.0 PL=0
MOVL C01044 V=800.0 PL=0
MOVL C01045 V=800.0 PL=0
MOVL C01046 V=800.0 PL=0
MOVL C01047 V=800.0 PL=0
MOVL C01048 V=800.0 PL=0
MOVL C01049 V=800.0 PL=0
MOVL C01050 V=800.0 PL=0
MOVL C01051 V=800.0 PL=0
MOVL C01052 V=800.0 PL=0
MOVL C01053 V=800.0 PL=0
MOVL C01054 V=800.0 PL=0
MOVL C01055 V=800.0 PL=0
MOVL C01056 V=800.0 PL=0
MOVL C01057 V=800.0 PL=0
MOVL C01058 V=800.0 PL=0
MOVL C01059 V=800.0 PL=0
MOVL C01060 V=800.0 PL=0
MOVL C01061 V=800.0 PL=0
MOVL C01062 V=800.0 PL=0
MOVL C01063 V=800.0 PL=0
MOVL C01064 V=800.0 PL=0
MOVL C01065 V=800.0 PL=0
MOVL C01066 V=800.0 PL=0
MOVL C01067 V=800.0 PL=0
MOVL C01068 V=800.0 PL=0
MOVL C01069 V=800.0 PL=0
MOVL C01070 V=800.0 PL=0
MOVL C01071 V=800.0 PL=0
MOVL C01072 V=800.0 PL=0
MOVL C01073 V=800.0 PL=0
MOVL C01074 V=800.0 PL=0
MOVL C01075 V=800.0 PL=0
MOVL C01076 V=800.0 PL=0
MOVL C01077 V=800.0 PL=0
MOVL C01078 V=800.0 PL=0
MOVL C01079 V=800.0 PL=0
MOVL C01080 V=800.0 PL=0
MOVL C01081 V=800.0 PL=0
MOVL C01082 V=800.0 PL=0
MOVL C01083 V=800.0 PL=0
MOVL C01084 V=800.0 PL=0
MOVL C01085 V=800.0 PL=0
MOVL C01086 V=800.0 PL=0
MOVL C01087 V=800.0 PL=0
MOVL C01088 V=800.0 PL=0
MOVL C01089 V=800.0 PL=0
MOVL C01090 V=800.0 PL=0
MOVL C01091 V=800.0 PL=0
MOVL C01092 V=800.0 PL=0
MOVL C01093 V=800.0 PL=0
MOVL C01094 V=800.0 PL=0
MOVL C01095 V=800.0 PL=0
MOVL C01096 V=800.0 PL=0
MOVL C01097 V=800.0 PL=0
MOVL C01098 V=800.0 PL=0
MOVL C01099 V=800.0 PL=0
MOVL C01100 V=800.0 PL=0
MOVL C01101 V=800.0 PL=0
MOVL C01102 V=800.0 PL=0
MOVL C01103 V=800.0 PL=0
MOVL C01104 V=800.0 PL=0
MOVL C01105 V=800.0 PL=0
MOVL C01106 V=800.0 PL=0
MOVL C01107 V=800.0 PL=0
MOVL C01108 V=800.0 PL=0
MOVL C01109 V=800.0 PL=0
MOVL C01110 V=800.0 PL=0
MOVL C01111 V=800.0 PL=0
MOVL C01112 V=800.0 PL=0
MOVL C01113 V=800.0 PL=0
MOVL C01114 V=800.0 PL=0
MOVL C01115 V=800.0 PL=0
MOVL C01116 V=800.0 PL=0
MOVL C01117 V=800.0 PL=0
MOVL C01118 V=800.0 PL=0
MOVL C01119 V=800.0 PL=0
MOVL C01120 V=800.0 PL=0
MOVL C01121 V=800.0 PL=0
MOVL C01122 V=800.0 PL=0
MOVL C01123 V=800.0 PL=0
MOVL C01124 V=800.0 PL=0
MOVL C01125 V=800.0 PL=0
MOVL C01126 V=800.0 PL=0
MOVL C01127 V=800.0 PL=0
MOVL C01128 V=800.0 PL=0
MOVL C01129 V=800.0 PL=0
MOVL C01130 V=800.0 PL=0
MOVL C01131 V=800.0 PL=0
MOVL C01132 V=800.0 PL=0
MOVL C01133 V=800.0 PL=0
MOVL C01134 V=800.0 PL=0
MOVL C01135 V=800.0 PL=0
MOVL C01136 V=800.0 PL=0
MOVL C01137 V=800.0 PL=0
MOVL C01138 V=800.0 PL=0
MOVL C01139 V=800.0 PL=0
MOVL C01140 V=800.0 PL=0
MOVL C01141 V=800.0 PL=0
MOVL C01142 V=800.0 PL=0
MOVL C01143 V=800.0 PL=0
MOVL C01144 V=800.0 PL=0
MOVL C01145 V=800.0 PL=0
MOVL C01146 V=800.0 PL=0
MOVL C01147 V=800.0 PL=0
MOVL C01148 V=800.0 PL=0
MOVL C01149 V=800.0 PL=0
MOVL C01150 V=800.0 PL=0
MOVL C01151 V=800.0 PL=0
MOVL C01152 V=800.0 PL=0
MOVL C01153 V=800.0 PL=0
MOVL C01154 V=800.0 PL=0
MOVL C01155 V=800.0 PL=0
MOVL C01156 V=800.0 PL=0
MOVL C01157 V=800.0 PL=0
MOVL C01158 V=800.0 PL=0
MOVL C01159 V=800.0 PL=0
MOVL C01160 V=800.0 PL=0
MOVL C01161 V=800.0 PL=0
MOVL C01162 V=800.0 PL=0
MOVL C01163 V=800.0 PL=0
MOVL C01164 V=800.0 PL=0
MOVL C01165 V=800.0 PL=0
MOVL C01166 V=800.0 PL=0
MOVL C01167 V=800.0 PL=0
MOVL C01168 V=800.0 PL=0
MOVL C01169 V=800.0 PL=0
MOVL C01170 V=800.0 PL=0
MOVL C01171 V=800.0 PL=0
MOVL C01172 V=800.0 PL=0
MOVL C01173 V=800.0 PL=0
MOVL C01174 V=800.0 PL=0
MOVL C01175 V=800.0 PL=0
MOVL C01176 V=800.0 PL=0
MOVL C01177 V=800.0 PL=0
MOVL C01178 V=800.0 PL=0
MOVL C01179 V=800.0 PL=0
MOVL C01180 V=800.0 PL=0
MOVL C01181 V=800.0 PL=0
MOVL C01182 V=800.0 PL=0
MOVL C01183 V=800.0 PL=0
MOVL C01184 V=800.0 PL=0
MOVL C01185 V=800.0 PL=0
MOVL C01186 V=800.0 PL=0
MOVL C01187 V=800.0 PL=0
MOVL C01188 V=800.0 PL=0
MOVL C01189 V=800.0 PL=0
MOVL C01190 V=800.0 PL=0
MOVL C01191 V=800.0 PL=0
MOVL C01192 V=800.0 PL=0
MOVL C01193 V=800.0 PL=0
MOVL C01194 V=800.0 PL=0
MOVL C01195 V=800.0 PL=0
MOVL C01196 V=800.0 PL=0
MOVL C01197 V=800.0 PL=0
MOVL C01198 V=800.0 PL=0
MOVL C01199 V=800.0 PL=0
MOVL C01200 V=800.0 PL=0
MOVL C01201 V=800.0 PL=0
MOVL C01202 V=800.0 PL=0
MOVL C01203 V=800.0 PL=0
MOVL C01204 V=800.0 PL=0
MOVL C01205 V=800.0 PL=0
MOVL C01206 V=800.0 PL=0
MOVL C01207 V=800.0 PL=0
MOVL C01208 V=800.0 PL=0
MOVL C01209 V=800.0 PL=0
MOVL C01210 V=800.0 PL=0
MOVL C01211 V=800.0 PL=0
MOVL C01212 V=800.0 PL=0
MOVL C01213 V=800.0 PL=0
MOVL C01214 V=800.0 PL=0
MOVL C01215 V=800.0 PL=0
MOVL C01216 V=800.0 PL=0
MOVL C01217 V=800.0 PL=0
MOVL C01218 V=800.0 PL=0
MOVL C01219 V=800.0 PL=0
MOVL C01220 V=800.0 PL=0
MOVL C01221 V=800.0 PL=0
MOVL C01222 V=800.0 PL=0
MOVL C01223 V=800.0 PL=0
MOVL C01224 V=800.0 PL=0
MOVL C01225 V=800.0 PL=0
MOVL C01226 V=800.0 PL=0
MOVL C01227 V=800.0 PL=0
MOVL C01228 V=800.0 PL=0
MOVL C01229 V=800.0 PL=0
MOVL C01230 V=800.0 PL=0
MOVL C01231 V=800.0 PL=0
MOVL C01232 V=800.0 PL=0
MOVL C01233 V=800.0 PL=0
MOVL C01234 V=800.0 PL=0
MOVL C01235 V=800.0 PL=0
MOVL C01236 V=800.0 PL=0
MOVL C01237 V=800.0 PL=0
MOVL C01238 V=800.0 PL=0
MOVL C01239 V=800.0 PL=0
MOVL C01240 V=800.0 PL=0
MOVL C01241 V=800.0 PL=0
MOVL C01242 V=800.0 PL=0
MOVL C01243 V=800.0 PL=0
MOVL C01244 V=800.0 PL=0
MOVL C01245 V=800.0 PL=0
MOVL C01246 V=800.0 PL=0
MOVL C01247 V=800.0 PL=0
MOVL C01248 V=800.0 PL=0
MOVL C01249 V=800.0 PL=0
MOVL C01250 V=800.0 PL=0
MOVL C01251 V=800.0 PL=0
MOVL C01252 V=800.0 PL=0
MOVL C01253 V=800.0 PL=0
MOVL C01254 V=800.0 PL=0
MOVL C01255 V=800.0 PL=0
MOVL C01256 V=800.0 PL=0
MOVL C01257 V=800.0 PL=0
MOVL C01258 V=800.0 PL=0
MOVL C01259 V=800.0 PL=0
MOVL C01260 V=800.0 PL=0
MOVL C01261 V=800.0 PL=0
MOVL C01262 V=800.0 PL=0
MOVL C01263 V=800.0 PL=0
MOVL C01264 V=800.0 PL=0
MOVL C01265 V=800.0 PL=0
MOVL C01266 V=800.0 PL=0
MOVL C01267 V=800.0 PL=0
MOVL C01268 V=800.0 PL=0
MOVL C01269 V=800.0 PL=0
MOVL C01270 V=800.0 PL=0
MOVL C01271 V=800.0 PL=0
MOVL C01272 V=800.0 PL=0
MOVL C01273 V=800.0 PL=0
MOVL C01274 V=800.0 PL=0
MOVL C01275 V=800.0 PL=0
MOVL C01276 V=800.0 PL=0
MOVL C01277 V=800.0 PL=0
MOVL C01278 V=800.0 PL=0
MOVL C01279 V=800.0 PL=0
MOVL C01280 V=800.0 PL=0
MOVL C01281 V=800.0 PL=0
MOVL C01282 V=800.0 PL=0
MOVL C01283 V=800.0 PL=0
MOVL C01284 V=800.0 PL=0
MOVL C01285 V=800.0 PL=0
MOVL C01286 V=800.0 PL=0
MOVL C01287 V=800.0 PL=0
MOVL C01288 V=800.0 PL=0
MOVL C01289 V=800.0 PL=0
MOVL C01290 V=800.0 PL=0
MOVL C01291 V=800.0 PL=0
MOVL C01292 V=800.0 PL=0
MOVL C01293 V=800.0 PL=0
MOVL C01294 V=800.0 PL=0
MOVL C01295 V=800.0 PL=0
MOVL C01296 V=800.0 PL=0
MOVL C01297 V=800.0 PL=0
MOVL C01298 V=800.0 PL=0
MOVL C01299 V=800.0 PL=0
MOVL C01300 V=800.0 PL=0
MOVL C01301 V=800.0 PL=0
MOVL C01302 V=800.0 PL=0
MOVL C01303 V=800.0 PL=0
MOVL C01304 V=800.0 PL=0
MOVL C01305 V=800.0 PL=0
MOVL C01306 V=800.0 PL=0
MOVL C01307 V=800.0 PL=0
MOVL C01308 V=800.0 PL=0
MOVL C01309 V=800.0 PL=0
MOVL C01310 V=800.0 PL=0
MOVL C01311 V=800.0 PL=0
MOVL C01312 V=800.0 PL=0
MOVL C01313 V=800.0 PL=0
MOVL C01314 V=800.0 PL=0
MOVL C01315 V=800.0 PL=0
MOVL C01316 V=800.0 PL=0
MOVL C01317 V=800.0 PL=0
MOVL C01318 V=800.0 PL=0
MOVL C01319 V=800.0 PL=0
MOVL C01320 V=800.0 PL=0
MOVL C01321 V=800.0 PL=0
MOVL C01322 V=800.0 PL=0
MOVL C01323 V=800.0 PL=0
MOVL C01324 V=800.0 PL=0
MOVL C01325 V=800.0 PL=0
MOVL C01326 V=800.0 PL=0
MOVL C01327 V=800.0 PL=0
MOVL C01328 V=800.0 PL=0
MOVL C01329 V=800.0 PL=0
MOVL C01330 V=800.0 PL=0
MOVL C01331 V=800.0 PL=0
MOVL C01332 V=800.0 PL=0
MOVL C01333 V=800.0 PL=0
MOVL C01334 V=800.0 PL=0
MOVL C01335 V=800.0 PL=0
MOVL C01336 V=800.0 PL=0
MOVL C01337 V=800.0 PL=0
MOVL C01338 V=800.0 PL=0
MOVL C01339 V=800.0 PL=0
MOVL C01340 V=800.0 PL=0
MOVL C01341 V=800.0 PL=0
MOVL C01342 V=800.0 PL=0
MOVL C01343 V=800.0 PL=0
MOVL C01344 V=800.0 PL=0
MOVL C01345 V=800.0 PL=0
MOVL C01346 V=800.0 PL=0
MOVL C01347 V=800.0 PL=0
MOVL C01348 V=800.0 PL=0
MOVL C01349 V=800.0 PL=0
MOVL C01350 V=800.0 PL=0
MOVL C01351 V=800.0 PL=0
MOVL C01352 V=800.0 PL=0
MOVL C01353 V=800.0 PL=0
MOVL C01354 V=800.0 PL=0
MOVL C01355 V=800.0 PL=0
MOVL C01356 V=800.0 PL=0
MOVL C01357 V=800.0 PL=0
MOVL C01358 V=800.0 PL=0
MOVL C01359 V=800.0 PL=0
MOVL C01360 V=800.0 PL=0
MOVL C01361 V=800.0 PL=0
MOVL C01362 V=800.0 PL=0
MOVL C01363 V=800.0 PL=0
MOVL C01364 V=800.0 PL=0
MOVL C01365 V=800.0 PL=0
MOVL C01366 V=800.0 PL=0
MOVL C01367 V=800.0 PL=0
MOVL C01368 V=800.0 PL=0
MOVL C01369 V=800.0 PL=0
MOVL C01370 V=800.0 PL=0
MOVL C01371 V=800.0 PL=0
MOVL C01372 V=800.0 PL=0
MOVL C01373 V=800.0 PL=0
MOVL C01374 V=800.0 PL=0
MOVL C01375 V=800.0 PL=0
MOVL C01376 V=800.0 PL=0
MOVL C01377 V=800.0 PL=0
MOVL C01378 V=800.0 PL=0
MOVL C01379 V=800.0 PL=0
MOVL C01380 V=800.0 PL=0
MOVL C01381 V=800.0 PL=0
MOVL C01382 V=800.0 PL=0
MOVL C01383 V=800.0 PL=0
MOVL C01384 V=800.0 PL=0
MOVL C01385 V=800.0 PL=0
MOVL C01386 V=800.0 PL=0
MOVL C01387 V=800.0 PL=0
MOVL C01388 V=800.0 PL=0
MOVL C01389 V=800.0 PL=0
MOVL C01390 V=800.0 PL=0
MOVL C01391 V=800.0 PL=0
MOVL C01392 V=800.0 PL=0
MOVL C01393 V=800.0 PL=0
MOVL C01394 V=800.0 PL=0
MOVL C01395 V=800.0 PL=0
MOVL C01396 V=800.0 PL=0
MOVL C01397 V=800.0 PL=0
MOVL C01398 V=800.0 PL=0
MOVL C01399 V=800.0 PL=0
MOVL C01400 V=800.0 PL=0
MOVL C01401 V=800.0 PL=0
MOVL C01402 V=800.0 PL=0
MOVL C01403 V=800.0 PL=0
MOVL C01404 V=800.0 PL=0
MOVL C01405 V=800.0 PL=0
MOVL C01406 V=800.0 PL=0
MOVL C01407 V=800.0 PL=0
MOVL C01408 V=800.0 PL=0
MOVL C01409 V=800.0 PL=0
MOVL C01410 V=800.0 PL=0
MOVL C01411 V=800.0 PL=0
MOVL C01412 V=800.0 PL=0
MOVL C01413 V=800.0 PL=0
MOVL C01414 V=800.0 PL=0
MOVL C01415 V=800.0 PL=0
MOVL C01416 V=800.0 PL=0
MOVL C01417 V=800.0 PL=0
MOVL C01418 V=800.0 PL=0
MOVL C01419 V=800.0 PL=0
MOVL C01420 V=800.0 PL=0
MOVL C01421 V=800.0 PL=0
MOVL C01422 V=800.0 PL=0
MOVL C01423 V=800.0 PL=0
MOVL C01424 V=800.0 PL=0
MOVL C01425 V=800.0 PL=0
MOVL C01426 V=800.0 PL=0
MOVL C01427 V=800.0 PL=0
MOVL C01428 V=800.0 PL=0
MOVL C01429 V=800.0 PL=0
MOVL C01430 V=800.0 PL=0
MOVL C01431 V=800.0 PL=0
MOVL C01432 V=800.0 PL=0
MOVL C01433 V=800.0 PL=0
MOVL C01434 V=800.0 PL=0
MOVL C01435 V=800.0 PL=0
MOVL C01436 V=800.0 PL=0
MOVL C01437 V=800.0 PL=0
MOVL C01438 V=800.0 PL=0
MOVL C01439 V=800.0 PL=0
MOVL C01440 V=800.0 PL=0
MOVL C01441 V=800.0 PL=0
MOVL C01442 V=800.0 PL=0
MOVL C01443 V=800.0 PL=0
MOVL C01444 V=800.0 PL=0
MOVL C01445 V=800.0 PL=0
MOVL C01446 V=800.0 PL=0
MOVL C01447 V=800.0 PL=0
MOVL C01448 V=800.0 PL=0
MOVL C01449 V=800.0 PL=0
MOVL C01450 V=800.0 PL=0
MOVL C01451 V=800.0 PL=0
MOVL C01452 V=800.0 PL=0
MOVL C01453 V=800.0 PL=0
MOVL C01454 V=800.0 PL=0
MOVL C01455 V=800.0 PL=0
MOVL C01456 V=800.0 PL=0
MOVL C01457 V=800.0 PL=0
MOVL C01458 V=800.0 PL=0
MOVL C01459 V=800.0 PL=0
MOVL C01460 V=800.0 PL=0
MOVL C01461 V=800.0 PL=0
MOVL C01462 V=800.0 PL=0
MOVL C01463 V=800.0 PL=0
MOVL C01464 V=800.0 PL=0
MOVL C01465 V=800.0 PL=0
MOVL C01466 V=800.0 PL=0
MOVL C01467 V=800.0 PL=0
MOVL C01468 V=800.0 PL=0
MOVL C01469 V=800.0 PL=0
MOVL C01470 V=800.0 PL=0
MOVL C01471 V=800.0 PL=0
MOVL C01472 V=800.0 PL=0
MOVL C01473 V=800.0 PL=0
MOVL C01474 V=800.0 PL=0
MOVL C01475 V=800.0 PL=0
MOVL C01476 V=800.0 PL=0
MOVL C01477 V=800.0 PL=0
MOVL C01478 V=800.0 PL=0
MOVL C01479 V=800.0 PL=0
MOVL C01480 V=800.0 PL=0
MOVL C01481 V=800.0 PL=0
MOVL C01482 V=800.0 PL=0
MOVL C01483 V=800.0 PL=0
MOVL C01484 V=800.0 PL=0
MOVL C01485 V=800.0 PL=0
MOVL C01486 V=800.0 PL=0
MOVL C01487 V=800.0 PL=0
MOVL C01488 V=800.0 PL=0
MOVL C01489 V=800.0 PL=0
MOVL C01490 V=800.0 PL=0
MOVL C01491 V=800.0 PL=0
MOVL C01492 V=800.0 PL=0
MOVL C01493 V=800.0 PL=0
MOVL C01494 V=800.0 PL=0
MOVL C01495 V=800.0 PL=0
MOVL C01496 V=800.0 PL=0
MOVL C01497 V=800.0 PL=0
MOVL C01498 V=800.0 PL=0
MOVL C01499 V=800.0 PL=0
MOVL C01500 V=800.0 PL=0
MOVL C01501 V=800.0 PL=0
MOVL C01502 V=800.0 PL=0
MOVL C01503 V=800.0 PL=0
MOVL C01504 V=800.0 PL=0
MOVL C01505 V=800.0 PL=0
MOVL C01506 V=800.0 PL=0
MOVL C01507 V=800.0 PL=0
MOVL C01508 V=800.0 PL=0
MOVL C01509 V=800.0 PL=0
MOVL C01510 V=800.0 PL=0
MOVL C01511 V=800.0 PL=0
MOVL C01512 V=800.0 PL=0
MOVL C01513 V=800.0 PL=0
MOVL C01514 V=800.0 PL=0
MOVL C01515 V=800.0 PL=0
MOVL C01516 V=800.0 PL=0
MOVL C01517 V=800.0 PL=0
MOVL C01518 V=800.0 PL=0
MOVL C01519 V=800.0 PL=0
MOVL C01520 V=800.0 PL=0
MOVL C01521 V=800.0 PL=0
MOVL C01522 V=800.0 PL=0
MOVL C01523 V=800.0 PL=0
MOVL C01524 V=800.0 PL=0
MOVL C01525 V=800.0 PL=0
MOVL C01526 V=800.0 PL=0
MOVL C01527 V=800.0 PL=0
MOVL C01528 V=800.0 PL=0
MOVL C01529 V=800.0 PL=0
MOVL C01530 V=800.0 PL=0
MOVL C01531 V=800.0 PL=0
MOVL C01532 V=800.0 PL=0
MOVL C01533 V=800.0 PL=0
MOVL C01534 V=800.0 PL=0
MOVL C01535 V=800.0 PL=0
MOVL C01536 V=800.0 PL=0
MOVL C01537 V=800.0 PL=0
MOVL C01538 V=800.0 PL=0
MOVL C01539 V=800.0 PL=0
MOVL C01540 V=800.0 PL=0
MOVL C01541 V=800.0 PL=0
MOVL C01542 V=800.0 PL=0
MOVL C01543 V=800.0 PL=0
MOVL C01544 V=800.0 PL=0
MOVL C01545 V=800.0 PL=0
MOVL C01546 V=800.0 PL=0
MOVL C01547 V=800.0 PL=0
MOVL C01548 V=800.0 PL=0
MOVL C01549 V=800.0 PL=0
MOVL C01550 V=800.0 PL=0
MOVL C01551 V=800.0 PL=0
MOVL C01552 V=800.0 PL=0
MOVL C01553 V=800.0 PL=0
MOVL C01554 V=800.0 PL=0
MOVL C01555 V=800.0 PL=0
MOVL C01556 V=800.0 PL=0
MOVL C01557 V=800.0 PL=0
MOVL C01558 V=800.0 PL=0
MOVL C01559 V=800.0 PL=0
MOVL C01560 V=800.0 PL=0
MOVL C01561 V=800.0 PL=0
MOVL C01562 V=800.0 PL=0
MOVL C01563 V=800.0 PL=0
MOVL C01564 V=800.0 PL=0
MOVL C01565 V=800.0 PL=0
MOVL C01566 V=800.0 PL=0
MOVL C01567 V=800.0 PL=0
MOVL C01568 V=800.0 PL=0
MOVL C01569 V=800.0 PL=0
MOVL C01570 V=800.0 PL=0
MOVL C01571 V=800.0 PL=0
MOVL C01572 V=800.0 PL=0
MOVL C01573 V=800.0 PL=0
MOVL C01574 V=800.0 PL=0
MOVL C01575 V=800.0 PL=0
MOVL C01576 V=800.0 PL=0
MOVL C01577 V=800.0 PL=0
MOVL C01578 V=800.0 PL=0
MOVL C01579 V=800.0 PL=0
MOVL C01580 V=800.0 PL=0
MOVL C01581 V=800.0 PL=0
MOVL C01582 V=800.0 PL=0
MOVL C01583 V=800.0 PL=0
MOVL C01584 V=800.0 PL=0
MOVL C01585 V=800.0 PL=0
MOVL C01586 V=800.0 PL=0
MOVL C01587 V=800.0 PL=0
MOVL C01588 V=800.0 PL=0
MOVL C01589 V=800.0 PL=0
MOVL C01590 V=800.0 PL=0
MOVL C01591 V=800.0 PL=0
MOVL C01592 V=800.0 PL=0
MOVL C01593 V=800.0 PL=0
MOVL C01594 V=800.0 PL=0
MOVL C01595 V=800.0 PL=0
MOVL C01596 V=800.0 PL=0
MOVL C01597 V=800.0 PL=0
MOVL C01598 V=800.0 PL=0
MOVL C01599 V=800.0 PL=0
MOVL C01600 V=800.0 PL=0
MOVL C01601 V=800.0 PL=0
MOVL C01602 V=800.0 PL=0
MOVL C01603 V=800.0 PL=0
MOVL C01604 V=800.0 PL=0
MOVL C01605 V=800.0 PL=0
MOVL C01606 V=800.0 PL=0
MOVL C01607 V=800.0 PL=0
MOVL C01608 V=800.0 PL=0
MOVL C01609 V=800.0 PL=0
MOVL C01610 V=800.0 PL=0
MOVL C01611 V=800.0 PL=0
MOVL C01612 V=800.0 PL=0
MOVL C01613 V=800.0 PL=0
MOVL C01614 V=800.0 PL=0
MOVL C01615 V=800.0 PL=0
MOVL C01616 V=800.0 PL=0
MOVL C01617 V=800.0 PL=0
MOVL C01618 V=800.0 PL=0
MOVL C01619 V=800.0 PL=0
MOVL C01620 V=800.0 PL=0
MOVL C01621 V=800.0 PL=0
MOVL C01622 V=800.0 PL=0
MOVL C01623 V=800.0 PL=0
MOVL C01624 V=800.0 PL=0
MOVL C01625 V=800.0 PL=0
MOVL C01626 V=800.0 PL=0
MOVL C01627 V=800.0 PL=0
MOVL C01628 V=800.0 PL=0
MOVL C01629 V=800.0 PL=0
MOVL C01630 V=800.0 PL=0
MOVL C01631 V=800.0 PL=0
MOVL C01632 V=800.0 PL=0
MOVL C01633 V=800.0 PL=0
MOVL C01634 V=800.0 PL=0
MOVL C01635 V=800.0 PL=0
MOVL C01636 V=800.0 PL=0
MOVL C01637 V=800.0 PL=0
MOVL C01638 V=800.0 PL=0
MOVL C01639 V=800.0 PL=0
MOVL C01640 V=800.0 PL=0
MOVL C01641 V=800.0 PL=0
MOVL C01642 V=800.0 PL=0
MOVL C01643 V=800.0 PL=0
MOVL C01644 V=800.0 PL=0
MOVL C01645 V=800.0 PL=0
MOVL C01646 V=800.0 PL=0
MOVL C01647 V=800.0 PL=0
MOVL C01648 V=800.0 PL=0
MOVL C01649 V=800.0 PL=0
MOVL C01650 V=800.0 PL=0
MOVL C01651 V=800.0 PL=0
MOVL C01652 V=800.0 PL=0
MOVL C01653 V=800.0 PL=0
MOVL C01654 V=800.0 PL=0
MOVL C01655 V=800.0 PL=0
MOVL C01656 V=800.0 PL=0
MOVL C01657 V=800.0 PL=0
MOVL C01658 V=800.0 PL=0
MOVL C01659 V=800.0 PL=0
MOVL C01660 V=800.0 PL=0
MOVL C01661 V=800.0 PL=0
MOVL C01662 V=800.0 PL=0
MOVL C01663 V=800.0 PL=0
MOVL C01664 V=800.0 PL=0
MOVL C01665 V=800.0 PL=0
MOVL C01666 V=800.0 PL=0
MOVL C01667 V=800.0 PL=0
MOVL C01668 V=800.0 PL=0
MOVL C01669 V=800.0 PL=0
MOVL C01670 V=800.0 PL=0
MOVL C01671 V=800.0 PL=0
MOVL C01672 V=800.0 PL=0
MOVL C01673 V=800.0 PL=0
MOVL C01674 V=800.0 PL=0
MOVL C01675 V=800.0 PL=0
MOVL C01676 V=800.0 PL=0
MOVL C01677 V=800.0 PL=0
MOVL C01678 V=800.0 PL=0
MOVL C01679 V=800.0 PL=0
MOVL C01680 V=800.0 PL=0
MOVL C01681 V=800.0 PL=0
MOVL C01682 V=800.0 PL=0
MOVL C01683 V=800.0 PL=0
MOVL C01684 V=800.0 PL=0
MOVL C01685 V=800.0 PL=0
MOVL C01686 V=800.0 PL=0
MOVL C01687 V=800.0 PL=0
MOVL C01688 V=800.0 PL=0
MOVL C01689 V=800.0 PL=0
MOVL C01690 V=800.0 PL=0
MOVL C01691 V=800.0 PL=0
MOVL C01692 V=800.0 PL=0
MOVL C01693 V=800.0 PL=0
MOVL C01694 V=800.0 PL=0
MOVL C01695 V=800.0 PL=0
MOVL C01696 V=800.0 PL=0
MOVL C01697 V=800.0 PL=0
MOVL C01698 V=800.0 PL=0
MOVL C01699 V=800.0 PL=0
MOVL C01700 V=800.0 PL=0
MOVL C01701 V=800.0 PL=0
MOVL C01702 V=800.0 PL=0
MOVL C01703 V=800.0 PL=0
MOVL C01704 V=800.0 PL=0
MOVL C01705 V=800.0 PL=0
MOVL C01706 V=800.0 PL=0
MOVL C01707 V=800.0 PL=0
MOVL C01708 V=800.0 PL=0
MOVL C01709 V=800.0 PL=0
MOVL C01710 V=800.0 PL=0
MOVL C01711 V=800.0 PL=0
MOVL C01712 V=800.0 PL=0
MOVL C01713 V=800.0 PL=0
MOVL C01714 V=800.0 PL=0
MOVL C01715 V=800.0 PL=0
MOVL C01716 V=800.0 PL=0
MOVL C01717 V=800.0 PL=0
MOVL C01718 V=800.0 PL=0
MOVL C01719 V=800.0 PL=0
MOVL C01720 V=800.0 PL=0
MOVL C01721 V=800.0 PL=0
MOVL C01722 V=800.0 PL=0
MOVL C01723 V=800.0 PL=0
MOVL C01724 V=800.0 PL=0
MOVL C01725 V=800.0 PL=0
MOVL C01726 V=800.0 PL=0
MOVL C01727 V=800.0 PL=0
MOVL C01728 V=800.0 PL=0
MOVL C01729 V=800.0 PL=0
MOVL C01730 V=800.0 PL=0
MOVL C01731 V=800.0 PL=0
MOVL C01732 V=800.0 PL=0
MOVL C01733 V=800.0 PL=0
MOVL C01734 V=800.0 PL=0
MOVL C01735 V=800.0 PL=0
MOVL C01736 V=800.0 PL=0
MOVL C01737 V=800.0 PL=0
MOVL C01738 V=800.0 PL=0
MOVL C01739 V=800.0 PL=0
MOVL C01740 V=800.0 PL=0
MOVL C01741 V=800.0 PL=0
MOVL C01742 V=800.0 PL=0
MOVL C01743 V=800.0 PL=0
MOVL C01744 V=800.0 PL=0
MOVL C01745 V=800.0 PL=0
MOVL C01746 V=800.0 PL=0
MOVL C01747 V=800.0 PL=0
MOVL C01748 V=800.0 PL=0
MOVL C01749 V=800.0 PL=0
MOVL C01750 V=800.0 PL=0
MOVL C01751 V=800.0 PL=0
MOVL C01752 V=800.0 PL=0
MOVL C01753 V=800.0 PL=0
MOVL C01754 V=800.0 PL=0
MOVL C01755 V=800.0 PL=0
MOVL C01756 V=800.0 PL=0
MOVL C01757 V=800.0 PL=0
MOVL C01758 V=800.0 PL=0
MOVL C01759 V=800.0 PL=0
MOVL C01760 V=800.0 PL=0
MOVL C01761 V=800.0 PL=0
MOVL C01762 V=800.0 PL=0
MOVL C01763 V=800.0 PL=0
MOVL C01764 V=800.0 PL=0
MOVL C01765 V=800.0 PL=0
MOVL C01766 V=800.0 PL=0
MOVL C01767 V=800.0 PL=0
MOVL C01768 V=800.0 PL=0
MOVL C01769 V=800.0 PL=0
MOVL C01770 V=800.0 PL=0
MOVL C01771 V=800.0 PL=0
MOVL C01772 V=800.0 PL=0
MOVL C01773 V=800.0 PL=0
MOVL C01774 V=800.0 PL=0
MOVL C01775 V=800.0 PL=0
MOVL C01776 V=800.0 PL=0
MOVL C01777 V=800.0 PL=0
MOVL C01778 V=800.0 PL=0
MOVL C01779 V=800.0 PL=0
MOVL C01780 V=800.0 PL=0
MOVL C01781 V=800.0 PL=0
MOVL C01782 V=800.0 PL=0
MOVL C01783 V=800.0 PL=0
MOVL C01784 V=800.0 PL=0
MOVL C01785 V=800.0 PL=0
MOVL C01786 V=800.0 PL=0
MOVL C01787 V=800.0 PL=0
MOVL C01788 V=800.0 PL=0
MOVL C01789 V=800.0 PL=0
MOVL C01790 V=800.0 PL=0
MOVL C01791 V=800.0 PL=0
MOVL C01792 V=800.0 PL=0
MOVL C01793 V=800.0 PL=0
MOVL C01794 V=800.0 PL=0
MOVL C01795 V=800.0 PL=0
MOVL C01796 V=800.0 PL=0
MOVL C01797 V=800.0 PL=0
MOVL C01798 V=800.0 PL=0
MOVL C01799 V=800.0 PL=0
MOVL C01800 V=800.0 PL=0
MOVL C01801 V=800.0 PL=0
MOVL C01802 V=800.0 PL=0
MOVL C01803 V=800.0 PL=0
MOVL C01804 V=800.0 PL=0
MOVL C01805 V=800.0 PL=0
MOVL C01806 V=800.0 PL=0
MOVL C01807 V=800.0 PL=0
MOVL C01808 V=800.0 PL=0
MOVL C01809 V=800.0 PL=0
MOVL C01810 V=800.0 PL=0
MOVL C01811 V=800.0 PL=0
MOVL C01812 V=800.0 PL=0
MOVL C01813 V=800.0 PL=0
MOVL C01814 V=800.0 PL=0
MOVL C01815 V=800.0 PL=0
MOVL C01816 V=800.0 PL=0
MOVL C01817 V=800.0 PL=0
MOVL C01818 V=800.0 PL=0
MOVL C01819 V=800.0 PL=0
MOVL C01820 V=800.0 PL=0
MOVL C01821 V=800.0 PL=0
MOVL C01822 V=800.0 PL=0
MOVL C01823 V=800.0 PL=0
MOVL C01824 V=800.0 PL=0
MOVL C01825 V=800.0 PL=0
MOVL C01826 V=800.0 PL=0
MOVL C01827 V=800.0 PL=0
MOVL C01828 V=800.0 PL=0
MOVL C01829 V=800.0 PL=0
MOVL C01830 V=800.0 PL=0
MOVL C01831 V=800.0 PL=0
MOVL C01832 V=800.0 PL=0
MOVL C01833 V=800.0 PL=0
MOVL C01834 V=800.0 PL=0
MOVL C01835 V=800.0 PL=0
MOVL C01836 V=800.0 PL=0
MOVL C01837 V=800.0 PL=0
MOVL C01838 V=800.0 PL=0
MOVL C01839 V=800.0 PL=0
MOVL C01840 V=800.0 PL=0
MOVL C01841 V=800.0 PL=0
MOVL C01842 V=800.0 PL=0
MOVL C01843 V=800.0 PL=0
MOVL C01844 V=800.0 PL=0
MOVL C01845 V=800.0 PL=0
MOVL C01846 V=800.0 PL=0
MOVL C01847 V=800.0 PL=0
MOVL C01848 V=800.0 PL=0
MOVL C01849 V=800.0 PL=0
MOVL C01850 V=800.0 PL=0
MOVL C01851 V=800.0 PL=0
MOVL C01852 V=800.0 PL=0
MOVL C01853 V=800.0 PL=0
MOVL C01854 V=800.0 PL=0
MOVL C01855 V=800.0 PL=0
MOVL C01856 V=800.0 PL=0
MOVL C01857 V=800.0 PL=0
MOVL C01858 V=800.0 PL=0
MOVL C01859 V=800.0 PL=0
MOVL C01860 V=800.0 PL=0
MOVL C01861 V=800.0 PL=0
MOVL C01862 V=800.0 PL=0
MOVL C01863 V=800.0 PL=0
MOVL C01864 V=800.0 PL=0
MOVL C01865 V=800.0 PL=0
MOVL C01866 V=800.0 PL=0
MOVL C01867 V=800.0 PL=0
MOVL C01868 V=800.0 PL=0
MOVL C01869 V=800.0 PL=0
MOVL C01870 V=800.0 PL=0
MOVL C01871 V=800.0 PL=0
MOVL C01872 V=800.0 PL=0
MOVL C01873 V=800.0 PL=0
MOVL C01874 V=800.0 PL=0
MOVL C01875 V=800.0 PL=0
MOVL C01876 V=800.0 PL=0
MOVL C01877 V=800.0 PL=0
MOVL C01878 V=800.0 PL=0
MOVL C01879 V=800.0 PL=0
MOVL C01880 V=800.0 PL=0
MOVL C01881 V=800.0 PL=0
MOVL C01882 V=800.0 PL=0
MOVL C01883 V=800.0 PL=0
MOVL C01884 V=800.0 PL=0
MOVL C01885 V=800.0 PL=0
MOVL C01886 V=800.0 PL=0
MOVL C01887 V=800.0 PL=0
MOVL C01888 V=800.0 PL=0
MOVL C01889 V=800.0 PL=0
MOVL C01890 V=800.0 PL=0
MOVL C01891 V=800.0 PL=0
MOVL C01892 V=800.0 PL=0
MOVL C01893 V=800.0 PL=0
MOVL C01894 V=800.0 PL=0
MOVL C01895 V=800.0 PL=0
MOVL C01896 V=800.0 PL=0
MOVL C01897 V=800.0 PL=0
MOVL C01898 V=800.0 PL=0
MOVL C01899 V=800.0 PL=0
MOVL C01900 V=800.0 PL=0
MOVL C01901 V=800.0 PL=0
MOVL C01902 V=800.0 PL=0
MOVL C01903 V=800.0 PL=0
MOVL C01904 V=800.0 PL=0
MOVL C01905 V=800.0 PL=0
MOVL C01906 V=800.0 PL=0
MOVL C01907 V=800.0 PL=0
MOVL C01908 V=800.0 PL=0
MOVL C01909 V=800.0 PL=0
MOVL C01910 V=800.0 PL=0
MOVL C01911 V=800.0 PL=0
MOVL C01912 V=800.0 PL=0
MOVL C01913 V=800.0 PL=0
MOVL C01914 V=800.0 PL=0
MOVL C01915 V=800.0 PL=0
MOVL C01916 V=800.0 PL=0
MOVL C01917 V=800.0 PL=0
MOVL C01918 V=800.0 PL=0
MOVL C01919 V=800.0 PL=0
MOVL C01920 V=800.0 PL=0
MOVL C01921 V=800.0 PL=0
MOVL C01922 V=800.0 PL=0
MOVL C01923 V=800.0 PL=0
MOVL C01924 V=800.0 PL=0
MOVL C01925 V=800.0 PL=0
MOVL C01926 V=800.0 PL=0
MOVL C01927 V=800.0 PL=0
MOVL C01928 V=800.0 PL=0
MOVL C01929 V=800.0 PL=0
MOVL C01930 V=800.0 PL=0
MOVL C01931 V=800.0 PL=0
MOVL C01932 V=800.0 PL=0
MOVL C01933 V=800.0 PL=0
MOVL C01934 V=800.0 PL=0
MOVL C01935 V=800.0 PL=0
MOVL C01936 V=800.0 PL=0
MOVL C01937 V=800.0 PL=0
MOVL C01938 V=800.0 PL=0
MOVL C01939 V=800.0 PL=0
MOVL C01940 V=800.0 PL=0
MOVL C01941 V=800.0 PL=0
MOVL C01942 V=800.0 PL=0
MOVL C01943 V=800.0 PL=0
MOVL C01944 V=800.0 PL=0
MOVL C01945 V=800.0 PL=0
MOVL C01946 V=800.0 PL=0
MOVL C01947 V=800.0 PL=0
MOVL C01948 V=800.0 PL=0
MOVL C01949 V=800.0 PL=0
MOVL C01950 V=800.0 PL=0
MOVL C01951 V=800.0 PL=0
MOVL C01952 V=800.0 PL=0
MOVL C01953 V=800.0 PL=0
MOVL C01954 V=800.0 PL=0
MOVL C01955 V=800.0 PL=0
MOVL C01956 V=800.0 PL=0
MOVL C01957 V=800.0 PL=0
MOVL C01958 V=800.0 PL=0
MOVL C01959 V=800.0 PL=0
MOVL C01960 V=800.0 PL=0
MOVL C01961 V=800.0 PL=0
MOVL C01962 V=800.0 PL=0
MOVL C01963 V=800.0 PL=0
MOVL C01964 V=800.0 PL=0
MOVL C01965 V=800.0 PL=0
MOVL C01966 V=800.0 PL=0
MOVL C01967 V=800.0 PL=0
MOVL C01968 V=800.0 PL=0
MOVL C01969 V=800.0 PL=0
MOVL C01970 V=800.0 PL=0
MOVL C01971 V=800.0 PL=0
MOVL C01972 V=800.0 PL=0
MOVL C01973 V=800.0 PL=0
MOVL C01974 V=800.0 PL=0
MOVL C01975 V=800.0 PL=0
MOVL C01976 V=800.0 PL=0
MOVL C01977 V=800.0 PL=0
MOVL C01978 V=800.0 PL=0
MOVL C01979 V=800.0 PL=0
MOVL C01980 V=800.0 PL=0
MOVL C01981 V=800.0 PL=0
MOVL C01982 V=800.0 PL=0
MOVL C01983 V=800.0 PL=0
MOVL C01984 V=800.0 PL=0
MOVL C01985 V=800.0 PL=0
MOVL C01986 V=800.0 PL=0
MOVL C01987 V=800.0 PL=0
MOVL C01988 V=800.0 PL=0
MOVL C01989 V=800.0 PL=0
MOVL C01990 V=800.0 PL=0
MOVL C01991 V=800.0 PL=0
MOVL C01992 V=800.0 PL=0
MOVL C01993 V=800.0 PL=0
MOVL C01994 V=800.0 PL=0
MOVL C01995 V=800.0 PL=0
MOVL C01996 V=800.0 PL=0
MOVL C01997 V=800.0 PL=0
MOVL C01998 V=800.0 PL=0
MOVL C01999 V=800.0 PL=0
MOVL C02000 V=800.0 PL=0
MOVL C02001 V=800.0 PL=0
MOVL C02002 V=800.0 PL=0
MOVL C02003 V=800.0 PL=0
MOVL C02004 V=800.0 PL=0
MOVL C02005 V=800.0 PL=0
MOVL C02006 V=800.0 PL=0
MOVL C02007 V=800.0 PL=0
MOVL C02008 V=800.0 PL=0
MOVL C02009 V=800.0 PL=0
MOVL C02010 V=800.0 PL=0
MOVL C02011 V=800.0 PL=0
MOVL C02012 V=800.0 PL=0
MOVL C02013 V=800.0 PL=0
MOVL C02014 V=800.0 PL=0
MOVL C02015 V=800.0 PL=0
MOVL C02016 V=800.0 PL=0
MOVL C02017 V=800.0 PL=0
MOVL C02018 V=800.0 PL=0
MOVL C02019 V=800.0 PL=0
MOVL C02020 V=800.0 PL=0
MOVL C02021 V=800.0 PL=0
MOVL C02022 V=800.0 PL=0
MOVL C02023 V=800.0 PL=0
MOVL C02024 V=800.0 PL=0
MOVL C02025 V=800.0 PL=0
MOVL C02026 V=800.0 PL=0
MOVL C02027 V=800.0 PL=0
MOVL C02028 V=800.0 PL=0
MOVL C02029 V=800.0 PL=0
MOVL C02030 V=800.0 PL=0
MOVL C02031 V=800.0 PL=0
MOVL C02032 V=800.0 PL=0
MOVL C02033 V=800.0 PL=0
MOVL C02034 V=800.0 PL=0
MOVL C02035 V=800.0 PL=0
MOVL C02036 V=800.0 PL=0
MOVL C02037 V=800.0 PL=0
